C09106=1036.501,256.965,387.007,171.006,42.916,158.201
C09107=1036.494,256.716,387.037,171.003,42.915,158.201
C09108=1036.487,256.469,387.066,171.000,42.914,158.200
C09109=1036.480,256.220,387.095,170.997,42.914,158.200
C09110=1036.474,255.973,387.125,170.993,42.913,158.200
C09111=1036.468,255.724,387.154,170.991,42.912,158.199
C09112=1036.461,255.476,387.183,170.987,42.911,158.199
C09113=1036.454,255.228,387.213,170.985,42.910,158.198
C09114=1036.447,254.979,387.242,170.981,42.910,158.198
C09115=1036.441,254.731,387.272,170.978,42.909,158.198
C09116=1036.433,254.483,387.301,170.976,42.908,158.197
C09117=1036.427,254.235,387.330,170.972,42.907,158.197
C09118=1036.420,253.987,387.360,170.969,42.907,158.196
C09119=1036.413,253.739,387.389,170.966,42.906,158.196
C09120=1036.407,253.490,387.419,170.963,42.905,158.196
C09121=1036.400,253.242,387.448,170.960,42.903,158.195
C09122=1036.394,252.994,387.477,170.957,42.903,158.195
C09123=1036.387,252.745,387.507,170.953,42.902,158.194
C09124=1036.380,252.498,387.535,170.951,42.901,158.194
C09125=1036.373,252.249,387.565,170.947,42.900,158.193
C09126=1036.367,252.001,387.594,170.945,42.899,158.193
C09127=1036.360,251.753,387.624,170.941,42.899,158.193
C09128=1036.353,251.504,387.653,170.938,42.898,158.192
C09129=1036.347,251.256,387.682,170.936,42.897,158.192
C09130=1036.340,251.009,387.711,170.932,42.896,158.191
C09131=1036.333,250.760,387.741,170.930,42.895,158.191
C09132=1036.327,250.512,387.770,170.926,42.895,158.191
C09133=1036.321,250.264,387.799,170.924,42.894,158.190
C09134=1036.314,250.015,387.828,170.920,42.893,158.190
C09135=1036.307,249.767,387.857,170.917,42.892,158.189
C09136=1036.301,249.519,387.887,170.914,42.891,158.189
C09137=1036.291,249.191,387.924,170.911,42.890,158.189
C09138=1036.283,248.864,387.963,170.906,42.889,158.188
C09139=1036.274,248.536,388.001,170.903,42.888,158.187
C09140=1036.266,248.209,388.040,170.899,42.887,158.187
C09141=1036.259,247.960,388.069,170.896,42.886,158.187
C09142=1036.253,247.712,388.098,170.892,42.885,158.186
C09143=1036.246,247.464,388.127,170.890,42.884,158.186
C09144=1036.240,247.216,388.156,170.886,42.884,158.185
C09145=1036.233,246.967,388.185,170.884,42.883,158.185
C09146=1036.226,246.719,388.214,170.880,42.882,158.185
C09147=1036.220,246.471,388.243,170.878,42.881,158.184
C09148=1036.214,246.223,388.272,170.874,42.880,158.184
C09149=1036.207,245.974,388.302,170.872,42.879,158.183
C09150=1036.200,245.726,388.330,170.869,42.879,158.183
C09151=1036.194,245.478,388.359,170.866,42.878,158.183
C09152=1036.188,245.230,388.388,170.863,42.877,158.182
C09153=1036.181,244.982,388.417,170.860,42.876,158.182
C09154=1036.174,244.733,388.447,170.858,42.875,158.181
C09155=1036.167,244.485,388.475,170.854,42.874,158.181
C09156=1036.161,244.237,388.504,170.852,42.874,158.181
C09157=1036.155,243.988,388.532,170.849,42.873,158.180
C09158=1036.148,243.740,388.561,170.846,42.873,158.180
C09159=1036.141,243.492,388.590,170.843,42.872,158.180
C09160=1036.134,243.244,388.619,170.840,42.871,158.179
C09161=1036.128,242.995,388.648,170.837,42.870,158.179
C09162=1036.122,242.747,388.676,170.834,42.869,158.178
C09163=1036.115,242.498,388.705,170.831,42.868,158.178
C09164=1036.108,242.250,388.734,170.829,42.868,158.178
C09165=1036.101,242.002,388.763,170.825,42.867,158.177
C09166=1036.095,241.754,388.790,170.823,42.867,158.177
C09167=1036.089,241.506,388.819,170.819,42.866,158.177
C09168=1036.082,241.258,388.848,170.817,42.865,158.176
C09169=1036.075,241.008,388.877,170.814,42.864,158.176
C09170=1036.068,240.761,388.905,170.811,42.863,158.175
C09171=1036.062,240.512,388.934,170.808,42.863,158.175
C09172=1036.055,240.264,388.962,170.805,42.862,158.175
C09173=1036.048,240.016,388.990,170.802,42.861,158.174
C09174=1036.042,239.767,389.018,170.800,42.861,158.174
C09175=1036.035,239.519,389.047,170.796,42.860,158.174
C09176=1036.028,239.271,389.076,170.794,42.860,158.173
C09177=1036.022,239.022,389.104,170.791,42.859,158.173
C09178=1036.015,238.775,389.133,170.788,42.858,158.173
C09179=1036.008,238.526,389.160,170.786,42.857,158.172
C09180=1036.002,238.278,389.189,170.782,42.857,158.172
C09181=1035.995,238.030,389.217,170.780,42.856,158.172
C09182=1035.987,237.781,389.246,170.776,42.855,158.171
C09183=1035.981,237.532,389.274,170.774,42.854,158.171
C09184=1035.974,237.284,389.303,170.771,42.854,158.170
C09185=1035.968,237.036,389.330,170.768,42.853,158.170
C09186=1035.961,236.788,389.358,170.766,42.852,158.170
C09187=1035.955,236.539,389.387,170.762,42.852,158.169
C09188=1035.948,236.291,389.415,170.760,42.851,158.169
C09189=1035.941,236.043,389.443,170.757,42.851,158.169
C09190=1035.935,235.795,389.471,170.754,42.850,158.168
C09191=1035.927,235.546,389.499,170.751,42.849,158.168
C09192=1035.921,235.297,389.528,170.749,42.849,158.168
C09193=1035.912,234.964,389.565,170.745,42.847,158.167
C09194=1035.903,234.631,389.603,170.742,42.846,158.167
C09195=1035.894,234.297,389.641,170.737,42.846,158.166
C09196=1035.885,233.964,389.679,170.734,42.845,158.166
C09197=1035.879,233.715,389.707,170.731,42.844,158.165
C09198=1035.872,233.467,389.735,170.728,42.844,158.165
C09199=1035.865,233.219,389.763,170.725,42.843,158.165
C09200=1035.859,232.970,389.791,170.723,42.842,158.164
C09201=1035.852,232.722,389.819,170.720,42.842,158.164
C09202=1035.846,232.474,389.848,170.717,42.841,158.164
C09203=1035.839,232.225,389.875,170.714,42.841,158.163
C09204=1035.832,231.977,389.903,170.712,42.840,158.163
C09205=1035.826,231.728,389.931,170.709,42.839,158.163
C09206=1035.819,231.481,389.959,170.706,42.838,158.162
C09207=1035.812,231.232,389.987,170.703,42.838,158.162
C09208=1035.806,230.983,390.015,170.701,42.837,158.162
C09209=1035.799,230.735,390.043,170.698,42.836,158.161
C09210=1035.793,230.487,390.071,170.695,42.836,158.161
C09211=1035.786,230.238,390.099,170.693,42.835,158.161
C09212=1035.779,229.990,390.126,170.690,42.835,158.160
C09213=1035.773,229.741,390.154,170.687,42.834,158.160
C09214=1035.766,229.493,390.183,170.685,42.833,158.160
C09215=1035.759,229.245,390.210,170.681,42.833,158.159
C09216=1035.752,228.997,390.238,170.679,42.832,158.159
C09217=1035.746,228.748,390.266,170.677,42.831,158.159
C09218=1035.739,228.500,390.293,170.673,42.831,158.158
C09219=1035.732,228.251,390.321,170.671,42.830,158.158
C09220=1035.726,228.003,390.349,170.669,42.829,158.158
C09221=1035.719,227.754,390.377,170.665,42.829,158.157
C09222=1035.712,227.506,390.404,170.663,42.828,158.157
C09223=1035.706,227.257,390.432,170.660,42.828,158.157
C09224=1035.699,227.009,390.460,170.657,42.827,158.156
C09225=1035.692,226.762,390.487,170.655,42.827,158.156
C09226=1035.685,226.513,390.514,170.651,42.826,158.156
C09227=1035.679,226.265,390.542,170.649,42.825,158.155
C09228=1035.672,226.016,390.569,170.647,42.825,158.155
C09229=1035.666,225.767,390.597,170.643,42.824,158.155
C09230=1035.659,225.519,390.625,170.641,42.824,158.154
C09231=1035.652,225.271,390.652,170.639,42.823,158.154
C09232=1035.645,225.022,390.679,170.636,42.822,158.154
C09233=1035.638,224.774,390.707,170.633,42.822,158.153
C09234=1035.631,224.525,390.735,170.631,42.821,158.153
C09235=1035.625,224.276,390.762,170.628,42.820,158.153
C09236=1035.618,224.028,390.790,170.625,42.820,158.153
C09237=1035.612,223.780,390.816,170.623,42.819,158.152
C09238=1035.605,223.532,390.844,170.620,42.818,158.152
C09239=1035.598,223.283,390.872,170.617,42.818,158.152
C09240=1035.592,223.035,390.900,170.615,42.817,158.151
C09241=1035.585,222.786,390.927,170.612,42.817,158.151
C09242=1035.579,222.538,390.954,170.610,42.816,158.151
C09243=1035.571,222.289,390.981,170.607,42.816,158.150
C09244=1035.565,222.042,391.009,170.604,42.815,158.150
C09245=1035.559,221.793,391.036,170.602,42.815,158.150
C09246=1035.552,221.544,391.064,170.600,42.814,158.149
C09247=1035.545,221.296,391.091,170.596,42.814,158.149
C09248=1035.538,221.048,391.118,170.594,42.813,158.149
C09249=1035.529,220.706,391.156,170.590,42.812,158.148
C09250=1035.520,220.365,391.194,170.587,42.811,158.148
C09251=1035.511,220.024,391.230,170.584,42.811,158.147
C09252=1035.502,219.684,391.268,170.580,42.809,158.147
C09253=1035.495,219.435,391.295,170.577,42.809,158.147
C09254=1035.489,219.186,391.322,170.574,42.809,158.146
C09255=1035.482,218.938,391.350,170.572,42.808,158.146
C09256=1035.475,218.689,391.377,170.570,42.808,158.146
C09257=1035.468,218.442,391.403,170.566,42.807,158.145
C09258=1035.462,218.192,391.430,170.564,42.806,158.145
C09259=1035.455,217.944,391.458,170.562,42.806,158.145
C09260=1035.448,217.695,391.485,170.559,42.805,158.145
C09261=1035.441,217.447,391.512,170.556,42.805,158.144
C09262=1035.435,217.199,391.538,170.554,42.804,158.144
C09263=1035.428,216.951,391.565,170.552,42.804,158.144
C09264=1035.421,216.702,391.592,170.549,42.803,158.143
C09265=1035.414,216.453,391.620,170.546,42.803,158.143
C09266=1035.408,216.205,391.646,170.543,42.802,158.143
C09267=1035.401,215.957,391.674,170.541,42.802,158.142
C09268=1035.394,215.708,391.700,170.539,42.801,158.142
C09269=1035.388,215.459,391.728,170.537,42.800,158.142
C09270=1035.381,215.211,391.754,170.533,42.800,158.142
C09271=1035.374,214.963,391.782,170.531,42.799,158.141
C09272=1035.367,214.714,391.808,170.529,42.799,158.141
C09273=1035.361,214.465,391.835,170.526,42.798,158.141
C09274=1035.354,214.218,391.862,170.524,42.798,158.140
C09275=1035.348,213.969,391.889,170.521,42.797,158.140
C09276=1035.341,213.720,391.916,170.518,42.797,158.140
C09277=1035.334,213.472,391.943,170.516,42.796,158.140
C09278=1035.327,213.223,391.969,170.514,42.796,158.139
C09279=1035.321,212.975,391.997,170.511,42.795,158.139
C09280=1035.314,212.726,392.024,170.508,42.794,158.139
C09281=1035.308,212.478,392.050,170.506,42.794,158.138
C09282=1035.300,212.230,392.077,170.503,42.793,158.138
C09283=1035.294,211.981,392.104,170.501,42.793,158.138
C09284=1035.287,211.733,392.130,170.499,42.792,158.137
C09285=1035.281,211.484,392.157,170.496,42.792,158.137
C09286=1035.274,211.235,392.185,170.493,42.791,158.137
C09287=1035.268,210.987,392.211,170.491,42.791,158.136
C09288=1035.261,210.738,392.238,170.489,42.790,158.136
C09289=1035.254,210.490,392.264,170.486,42.789,158.136
C09290=1035.248,210.242,392.291,170.484,42.789,158.136
C09291=1035.240,209.993,392.318,170.482,42.789,158.135
C09292=1035.233,209.744,392.344,170.478,42.788,158.135
C09293=1035.228,209.496,392.371,170.476,42.788,158.135
C09294=1035.220,209.247,392.397,170.474,42.787,158.134
C09295=1035.214,208.999,392.423,170.471,42.787,158.134
C09296=1035.207,208.751,392.451,170.469,42.786,158.134
C09297=1035.200,208.502,392.477,170.467,42.785,158.134
C09298=1035.194,208.254,392.504,170.464,42.785,158.133
C09299=1035.187,208.005,392.530,170.461,42.785,158.133
C09300=1035.180,207.756,392.557,170.459,42.784,158.133
C09301=1035.174,207.508,392.583,170.456,42.784,158.133
C09302=1035.167,207.259,392.609,170.454,42.783,158.132
C09303=1035.160,207.011,392.635,170.452,42.782,158.132
C09304=1035.154,206.762,392.663,170.450,42.782,158.132
C09305=1035.144,206.427,392.698,170.446,42.781,158.131
C09306=1035.135,206.092,392.733,170.443,42.781,158.131
C09307=1035.125,205.756,392.769,170.439,42.781,158.131
C09308=1035.117,205.421,392.805,170.436,42.780,158.130
C09309=1035.090,204.371,392.911,170.114,42.675,158.085
C09310=1035.085,204.123,392.935,170.111,42.676,158.085
C09311=1035.079,203.874,392.961,170.108,42.675,158.085
C09312=1035.073,203.625,392.986,170.105,42.676,158.085
C09313=1035.066,203.377,393.011,170.101,42.677,158.085
C09314=1035.059,203.128,393.036,170.097,42.676,158.084
C09315=1035.054,202.879,393.061,170.094,42.677,158.084
C09316=1035.048,202.631,393.086,170.091,42.677,158.084
C09317=1035.042,202.382,393.111,170.088,42.677,158.084
C09318=1035.036,202.133,393.136,170.084,42.678,158.084
C09319=1035.030,201.884,393.161,170.081,42.678,158.083
C09320=1035.023,201.636,393.186,170.078,42.678,158.083
C09321=1035.018,201.388,393.211,170.075,42.678,158.083
C09322=1035.012,201.138,393.236,170.071,42.679,158.083
C09323=1035.005,200.890,393.261,170.067,42.679,158.083
C09324=1034.999,200.641,393.285,170.064,42.679,158.083
C09325=1034.993,200.392,393.311,170.061,42.680,158.082
C09326=1034.987,200.144,393.334,170.058,42.680,158.082
C09327=1034.981,199.895,393.360,170.054,42.681,158.082
C09328=1034.974,199.647,393.384,170.051,42.681,158.082
C09329=1034.968,199.397,393.409,170.048,42.681,158.082
C09330=1034.962,199.148,393.434,170.045,42.682,158.082
C09331=1034.956,198.901,393.458,170.042,42.682,158.082
C09332=1034.950,198.651,393.483,170.038,42.683,158.081
C09333=1034.943,198.403,393.507,170.035,42.683,158.081
C09334=1034.937,198.154,393.532,170.031,42.683,158.081
C09335=1034.930,197.905,393.557,170.028,42.683,158.081
C09336=1034.925,197.657,393.581,170.025,42.684,158.081
C09337=1034.918,197.408,393.606,170.021,42.685,158.081
C09338=1034.912,197.159,393.630,170.018,42.685,158.080
C09339=1034.905,196.910,393.654,170.015,42.686,158.080
C09340=1034.899,196.662,393.679,170.012,42.685,158.080
C09341=1034.893,196.413,393.703,170.009,42.686,158.080
C09342=1034.887,196.164,393.728,170.005,42.687,158.080
C09343=1034.881,195.916,393.752,170.002,42.687,158.080
C09344=1034.875,195.667,393.777,169.999,42.688,158.080
C09345=1034.868,195.418,393.801,169.996,42.688,158.079
C09346=1034.862,195.170,393.826,169.993,42.689,158.079
C09347=1034.856,194.921,393.850,169.990,42.689,158.079
C09348=1034.850,194.672,393.875,169.985,42.689,158.079
C09349=1034.844,194.424,393.900,169.982,42.690,158.079
C09350=1034.838,194.175,393.924,169.979,42.690,158.079
C09351=1034.832,193.925,393.948,169.976,42.691,158.079
C09352=1034.826,193.677,393.972,169.973,42.691,158.078
C09353=1034.819,193.428,393.997,169.970,42.692,158.078
C09354=1034.813,193.179,394.021,169.967,42.692,158.078
C09355=1034.808,192.931,394.046,169.963,42.693,158.078
C09356=1034.801,192.682,394.070,169.960,42.693,158.078
C09357=1034.795,192.433,394.094,169.957,42.694,158.078
C09358=1034.789,192.185,394.119,169.954,42.693,158.078
C09359=1034.783,191.936,394.143,169.951,42.694,158.077
C09360=1034.777,191.687,394.167,169.948,42.694,158.077
C09361=1034.770,191.438,394.191,169.945,42.695,158.077
C09362=1034.765,191.190,394.215,169.942,42.695,158.077
C09363=1034.758,190.941,394.239,169.939,42.696,158.077
C09364=1034.752,190.692,394.264,169.935,42.697,158.077
C09365=1034.746,190.444,394.288,169.932,42.697,158.077
C09366=1034.740,190.195,394.313,169.928,42.698,158.077
C09367=1034.734,189.946,394.336,169.925,42.698,158.076
C09368=1034.728,189.697,394.361,169.922,42.699,158.076
C09369=1034.722,189.449,394.385,169.919,42.699,158.076
C09370=1034.715,189.165,394.413,169.915,42.700,158.076
C09371=1034.708,188.880,394.440,169.912,42.700,158.076
C09372=1034.701,188.597,394.468,169.909,42.701,158.076
C09373=1034.694,188.312,394.495,169.905,42.701,158.076
C09374=1034.689,188.063,394.519,169.902,42.702,158.076
C09375=1034.682,187.814,394.543,169.899,42.702,158.075
C09376=1034.677,187.566,394.567,169.896,42.702,158.075
C09377=1034.671,187.317,394.591,169.893,42.703,158.075
C09378=1034.665,187.068,394.616,169.890,42.703,158.075
C09379=1034.659,186.819,394.640,169.887,42.704,158.075
C09380=1034.653,186.571,394.664,169.884,42.704,158.075
C09381=1034.647,186.322,394.688,169.881,42.705,158.075
C09382=1034.641,186.073,394.712,169.878,42.705,158.074
C09383=1034.635,185.825,394.736,169.875,42.706,158.074
C09384=1034.629,185.576,394.760,169.872,42.706,158.074
C09385=1034.623,185.327,394.784,169.869,42.707,158.074
C09386=1034.617,185.078,394.808,169.865,42.707,158.074
C09387=1034.611,184.830,394.833,169.862,42.708,158.074
C09388=1034.605,184.582,394.856,169.859,42.708,158.074
C09389=1034.600,184.332,394.880,169.856,42.709,158.074
C09390=1034.594,184.083,394.904,169.853,42.709,158.073
C09391=1034.588,183.834,394.928,169.850,42.709,158.073
C09392=1034.582,183.586,394.952,169.847,42.710,158.073
C09393=1034.576,183.338,394.976,169.844,42.710,158.073
C09394=1034.570,183.088,395.000,169.841,42.712,158.073
C09395=1034.564,182.839,395.023,169.838,42.712,158.073
C09396=1034.557,182.591,395.047,169.834,42.713,158.073
C09397=1034.551,182.342,395.070,169.831,42.713,158.073
C09398=1034.544,182.093,395.094,169.828,42.714,158.073
C09399=1034.539,181.844,395.117,169.825,42.715,158.073
C09400=1034.532,181.595,395.141,169.822,42.715,158.073
C09401=1034.526,181.347,395.164,169.819,42.716,158.073
C09402=1034.520,181.097,395.188,169.816,42.717,158.072
C09403=1034.514,180.849,395.211,169.813,42.717,158.072
C09404=1034.507,180.600,395.234,169.811,42.719,158.072
C09405=1034.501,180.351,395.258,169.808,42.719,158.072
C09406=1034.495,180.102,395.281,169.804,42.720,158.072
C09407=1034.488,179.853,395.305,169.802,42.721,158.072
C09408=1034.482,179.604,395.328,169.799,42.721,158.072
C09409=1034.476,179.356,395.351,169.796,42.722,158.072
C09410=1034.470,179.107,395.375,169.793,42.723,158.072
C09411=1034.463,178.859,395.398,169.790,42.723,158.072
C09412=1034.457,178.609,395.421,169.787,42.724,158.072
C09413=1034.451,178.361,395.445,169.784,42.725,158.072
C09414=1034.445,178.112,395.468,169.781,42.725,158.072
C09415=1034.439,177.863,395.492,169.778,42.727,158.072
C09416=1034.433,177.614,395.515,169.775,42.727,158.072
C09417=1034.426,177.365,395.537,169.772,42.728,158.071
C09418=1034.420,177.116,395.561,169.769,42.729,158.071
C09419=1034.414,176.867,395.584,169.766,42.729,158.071
C09420=1034.408,176.619,395.608,169.763,42.730,158.071
C09421=1034.402,176.370,395.631,169.760,42.731,158.071
C09422=1034.396,176.121,395.654,169.757,42.731,158.071
C09423=1034.390,175.872,395.677,169.754,42.732,158.071
C09424=1034.383,175.623,395.700,169.751,42.733,158.071
C09425=1034.377,175.374,395.723,169.748,42.733,158.071
C09426=1034.371,175.126,395.747,169.745,42.735,158.071
C09427=1034.365,174.876,395.770,169.742,42.735,158.071
C09428=1034.359,174.627,395.793,169.739,42.735,158.071
C09429=1034.353,174.379,395.817,169.736,42.737,158.071
C09430=1034.346,174.131,395.839,169.733,42.737,158.071
C09431=1034.340,173.881,395.862,169.730,42.738,158.071
C09432=1034.334,173.633,395.886,169.727,42.739,158.070
C09433=1034.328,173.384,395.909,169.724,42.739,158.070
C09434=1034.321,173.099,395.935,169.722,42.740,158.070
C09435=1034.314,172.815,395.962,169.718,42.741,158.070
C09436=1034.308,172.530,395.988,169.715,42.742,158.070
C09437=1034.300,172.246,396.014,169.712,42.743,158.070
C09438=1034.295,171.997,396.037,169.709,42.744,158.070
C09439=1034.288,171.748,396.060,169.706,42.744,158.070
C09440=1034.282,171.499,396.084,169.703,42.745,158.070
C09441=1034.276,171.251,396.106,169.700,42.746,158.070
C09442=1034.270,171.002,396.129,169.697,42.746,158.070
C09443=1034.264,170.753,396.152,169.694,42.748,158.070
C09444=1034.258,170.503,396.176,169.691,42.748,158.070
C09445=1034.252,170.255,396.198,169.688,42.749,158.070
C09446=1034.246,170.006,396.222,169.685,42.750,158.070
C09447=1034.240,169.758,396.244,169.682,42.750,158.069
C09448=1034.234,169.509,396.267,169.680,42.751,158.070
C09449=1034.228,169.260,396.290,169.677,42.752,158.069
C09450=1034.222,169.010,396.314,169.674,42.752,158.069
C09451=1034.215,168.762,396.336,169.671,42.753,158.069
C09452=1034.210,168.513,396.359,169.668,42.754,158.069
C09453=1034.204,168.264,396.382,169.665,42.755,158.069
C09454=1034.198,168.015,396.405,169.662,42.755,158.069
C09455=1034.193,167.766,396.428,169.659,42.756,158.069
C09456=1034.186,167.518,396.450,169.656,42.757,158.069
C09457=1034.180,167.269,396.474,169.654,42.757,158.069
C09458=1034.174,167.020,396.497,169.652,42.758,158.069
C09459=1034.168,166.771,396.520,169.649,42.759,158.069
C09460=1034.162,166.522,396.543,169.646,42.760,158.069
C09461=1034.156,166.273,396.565,169.643,42.761,158.069
C09462=1034.150,166.024,396.588,169.640,42.761,158.069
C09463=1034.144,165.776,396.611,169.637,42.762,158.069
C09464=1034.139,165.527,396.634,169.635,42.763,158.069
C09465=1034.132,165.278,396.657,169.632,42.764,158.069
C09466=1034.127,165.029,396.679,169.629,42.764,158.068
C09467=1034.121,164.780,396.702,169.626,42.765,158.068
C09468=1034.115,164.531,396.725,169.623,42.766,158.068
C09469=1034.110,164.282,396.748,169.620,42.766,158.068
C09470=1034.103,164.033,396.770,169.618,42.767,158.068
C09471=1034.097,163.784,396.793,169.615,42.768,158.068
C09472=1034.092,163.535,396.816,169.612,42.769,158.068
C09473=1034.086,163.287,396.839,169.609,42.769,158.068
C09474=1034.079,163.038,396.861,169.606,42.770,158.068
C09475=1034.074,162.789,396.884,169.604,42.771,158.068
C09476=1034.068,162.540,396.907,169.601,42.771,158.068
C09477=1034.063,162.291,396.929,169.599,42.772,158.068
C09478=1034.056,162.042,396.952,169.595,42.773,158.068
C09479=1034.050,161.793,396.975,169.593,42.774,158.068
C09480=1034.045,161.544,396.998,169.591,42.774,158.068
C09481=1034.039,161.295,397.020,169.588,42.776,158.068
C09482=1034.032,161.047,397.043,169.585,42.776,158.068
C09483=1034.027,160.797,397.065,169.582,42.777,158.068
C09484=1034.021,160.548,397.088,169.579,42.778,158.067
C09485=1034.015,160.300,397.111,169.577,42.778,158.067
C09486=1034.009,160.051,397.133,169.574,42.779,158.067
C09487=1034.004,159.801,397.156,169.571,42.780,158.067
C09488=1033.997,159.553,397.178,169.568,42.781,158.067
C09489=1033.991,159.304,397.201,169.565,42.782,158.067
C09490=1033.985,159.055,397.222,169.563,42.782,158.067
C09491=1033.979,158.806,397.245,169.560,42.783,158.067
C09492=1033.973,158.557,397.268,169.558,42.785,158.067
C09493=1033.967,158.308,397.289,169.554,42.785,158.067
C09494=1033.960,158.059,397.312,169.552,42.786,158.067
C09495=1033.955,157.810,397.334,169.549,42.787,158.067
C09496=1033.949,157.561,397.356,169.547,42.788,158.067
C09497=1033.942,157.312,397.378,169.544,42.789,158.067
C09498=1033.935,157.028,397.404,169.541,42.790,158.067
C09499=1033.929,156.743,397.429,169.537,42.791,158.067
C09500=1033.922,156.458,397.454,169.534,42.792,158.067
C09501=1033.915,156.173,397.480,169.531,42.793,158.067
C09502=1033.908,155.924,397.502,169.529,42.794,158.067
C09503=1033.903,155.675,397.525,169.525,42.794,158.067
C09504=1033.897,155.426,397.546,169.524,42.795,158.067
C09505=1033.891,155.178,397.569,169.521,42.797,158.067
C09506=1033.885,154.928,397.591,169.518,42.797,158.067
C09507=1033.879,154.680,397.613,169.515,42.798,158.067
C09508=1033.873,154.430,397.635,169.512,42.799,158.067
C09509=1033.867,154.182,397.658,169.510,42.800,158.067
C09510=1033.861,153.932,397.679,169.507,42.801,158.067
C09511=1033.854,153.683,397.701,169.504,42.802,158.067
C09512=1033.848,153.435,397.723,169.502,42.803,158.067
C09513=1033.842,153.185,397.745,169.499,42.804,158.067
C09514=1033.836,152.936,397.768,169.497,42.805,158.067
C09515=1033.831,152.688,397.789,169.494,42.806,158.067
C09516=1033.824,152.439,397.811,169.491,42.807,158.067
C09517=1033.818,152.190,397.833,169.488,42.807,158.067
C09518=1033.812,151.941,397.855,169.485,42.808,158.067
C09519=1033.806,151.692,397.876,169.483,42.809,158.067
C09520=1033.800,151.443,397.899,169.480,42.811,158.067
C09521=1033.794,151.194,397.921,169.477,42.811,158.067
C09522=1033.788,150.944,397.943,169.475,42.812,158.067
C09523=1033.782,150.697,397.965,169.473,42.813,158.067
C09524=1033.776,150.447,397.986,169.470,42.814,158.067
C09525=1033.769,150.198,398.008,169.467,42.815,158.067
C09526=1033.764,149.949,398.030,169.464,42.816,158.067
C09527=1033.757,149.700,398.052,169.462,42.817,158.067
C09528=1033.751,149.451,398.074,169.459,42.818,158.067
C09529=1033.746,149.202,398.095,169.456,42.819,158.067
C09530=1033.740,148.953,398.117,169.453,42.820,158.067
C09531=1033.733,148.705,398.139,169.452,42.821,158.067
C09532=1033.727,148.455,398.161,169.449,42.822,158.067
C09533=1033.721,148.206,398.183,169.446,42.822,158.067
C09534=1033.715,147.958,398.204,169.443,42.823,158.067
C09535=1033.710,147.708,398.226,169.441,42.824,158.067
C09536=1033.704,147.459,398.248,169.438,42.826,158.067
C09537=1033.697,147.210,398.270,169.435,42.827,158.067
C09538=1033.691,146.961,398.292,169.432,42.827,158.067
C09539=1033.685,146.713,398.313,169.431,42.828,158.067
C09540=1033.679,146.463,398.335,169.428,42.829,158.067
C09541=1033.673,146.214,398.356,169.425,42.831,158.067
C09542=1033.667,145.965,398.378,169.422,42.832,158.067
C09543=1033.660,145.716,398.399,169.420,42.833,158.067
C09544=1033.654,145.468,398.420,169.417,42.833,158.067
C09545=1033.648,145.218,398.442,169.414,42.834,158.067
C09546=1033.642,144.969,398.464,169.411,42.835,158.067
C09547=1033.636,144.720,398.485,169.410,42.836,158.067
C09548=1033.630,144.471,398.507,169.407,42.838,158.067
C09549=1033.624,144.222,398.528,169.404,42.839,158.067
C09550=1033.618,143.973,398.550,169.401,42.840,158.067
C09551=1033.612,143.724,398.571,169.399,42.841,158.067
C09552=1033.605,143.475,398.592,169.396,42.841,158.067
C09553=1033.599,143.226,398.614,169.393,42.842,158.067
C09554=1033.593,142.977,398.635,169.392,42.843,158.067
C09555=1033.587,142.728,398.657,169.389,42.845,158.067
C09556=1033.581,142.479,398.679,169.386,42.846,158.067
C09557=1033.575,142.230,398.700,169.383,42.847,158.067
C09558=1033.569,141.981,398.721,169.381,42.848,158.067
C09559=1033.563,141.732,398.743,169.378,42.848,158.067
C09560=1033.558,141.483,398.764,169.375,42.849,158.067
C09561=1033.551,141.235,398.785,169.374,42.850,158.067
C09562=1033.543,140.886,398.815,169.370,42.852,158.067
C09563=1033.534,140.536,398.846,169.366,42.854,158.067
C09564=1033.525,140.188,398.875,169.362,42.855,158.067
C09565=1033.517,139.839,398.905,169.358,42.856,158.067
C09566=1033.511,139.590,398.926,169.356,42.857,158.067
C09567=1033.505,139.341,398.948,169.354,42.858,158.067
C09568=1033.499,139.092,398.969,169.351,42.860,158.067
C09569=1033.493,138.843,398.991,169.349,42.861,158.067
C09570=1033.486,138.594,399.012,169.346,42.861,158.067
C09571=1033.481,138.345,399.033,169.343,42.862,158.067
C09572=1033.475,138.096,399.054,169.341,42.863,158.067
C09573=1033.468,137.847,399.075,169.338,42.864,158.067
C09574=1033.462,137.598,399.097,169.336,42.866,158.067
C09575=1033.457,137.348,399.117,169.333,42.867,158.067
C09576=1033.450,137.100,399.138,169.331,42.868,158.067
C09577=1033.444,136.851,399.160,169.328,42.869,158.067
C09578=1033.438,136.602,399.181,169.325,42.870,158.067
C09579=1033.433,136.353,399.202,169.323,42.871,158.067
C09580=1033.426,136.104,399.223,169.321,42.872,158.067
C09581=1033.420,135.855,399.245,169.318,42.873,158.067
C09582=1033.414,135.606,399.265,169.316,42.874,158.067
C09583=1033.408,135.357,399.286,169.313,42.875,158.067
C09584=1033.401,135.107,399.308,169.310,42.876,158.067
C09585=1033.395,134.859,399.328,169.308,42.877,158.067
C09586=1033.389,134.609,399.349,169.306,42.879,158.067
C09587=1033.384,134.360,399.370,169.303,42.880,158.067
C09588=1033.377,134.111,399.391,169.301,42.881,158.068
C09589=1033.371,133.862,399.413,169.298,42.882,158.068
C09590=1033.365,133.613,399.433,169.295,42.883,158.068
C09591=1033.359,133.364,399.454,169.293,42.884,158.068
C09592=1033.353,133.115,399.475,169.291,42.885,158.068
C09593=1033.347,132.866,399.496,169.288,42.886,158.068
C09594=1033.340,132.617,399.517,169.286,42.887,158.068
C09595=1033.334,132.368,399.537,169.283,42.888,158.068
C09596=1033.328,132.119,399.559,169.280,42.890,158.068
C09597=1033.323,131.870,399.580,169.278,42.890,158.068
C09598=1033.316,131.621,399.601,169.275,42.891,158.068
C09599=1033.311,131.372,399.621,169.272,42.892,158.068
C09600=1033.304,131.123,399.642,169.271,42.893,158.068
C09601=1033.299,130.874,399.663,169.268,42.894,158.068
C09602=1033.293,130.625,399.684,169.265,42.896,158.068
C09603=1033.286,130.375,399.705,169.263,42.896,158.068
C09604=1033.280,130.127,399.725,169.260,42.898,158.068
C09605=1033.273,129.877,399.746,169.258,42.899,158.068
C09606=1033.268,129.628,399.766,169.256,42.900,158.068
C09607=1033.261,129.379,399.787,169.253,42.902,158.068
C09608=1033.255,129.131,399.807,169.250,42.903,158.068
C09609=1033.249,128.881,399.829,169.248,42.904,158.068
C09610=1033.242,128.632,399.849,169.245,42.905,158.068
C09611=1033.236,128.383,399.869,169.243,42.906,158.068
C09612=1033.229,128.134,399.890,169.240,42.908,158.068
C09613=1033.224,127.885,399.911,169.238,42.909,158.068
C09614=1033.217,127.635,399.931,169.235,42.910,158.068
C09615=1033.211,127.387,399.952,169.232,42.911,158.068
C09616=1033.205,127.137,399.973,169.231,42.912,158.068
C09617=1033.199,126.889,399.993,169.228,42.913,158.068
C09618=1033.192,126.640,400.014,169.225,42.914,158.068
C09619=1033.186,126.391,400.034,169.223,42.915,158.069
C09620=1033.180,126.141,400.055,169.221,42.917,158.069
C09621=1033.174,125.892,400.075,169.218,42.918,158.069
C09622=1033.165,125.521,400.105,169.215,42.919,158.069
C09623=1033.156,125.150,400.136,169.211,42.921,158.069
C09624=1033.149,124.865,400.160,169.208,42.923,158.069
C09625=1033.142,124.579,400.183,169.205,42.924,158.069
C09626=1033.135,124.295,400.206,169.203,42.926,158.069
C09627=1033.128,124.010,400.230,169.199,42.927,158.069
C09628=1033.122,123.760,400.251,169.197,42.928,158.069
C09629=1033.116,123.511,400.271,169.194,42.929,158.069
C09630=1033.109,123.261,400.291,169.193,42.930,158.069
C09631=1033.103,123.013,400.312,169.190,42.931,158.069
C09632=1033.097,122.763,400.332,169.187,42.932,158.069
C09633=1033.091,122.515,400.352,169.185,42.934,158.069
C09634=1033.085,122.266,400.372,169.182,42.935,158.069
C09635=1033.078,122.016,400.393,169.180,42.936,158.069
C09636=1033.073,121.767,400.413,169.178,42.937,158.069
C09637=1033.067,121.518,400.434,169.175,42.938,158.069
C09638=1033.060,121.269,400.454,169.173,42.939,158.069
C09639=1033.054,121.021,400.474,169.170,42.941,158.069
C09640=1033.048,120.771,400.495,169.167,42.942,158.070
C09641=1033.042,120.522,400.515,169.166,42.943,158.070
C09642=1033.036,120.272,400.535,169.163,42.944,158.070
C09643=1033.030,120.024,400.555,169.161,42.945,158.070
C09644=1033.025,119.774,400.576,169.158,42.947,158.070
C09645=1033.018,119.525,400.596,169.155,42.948,158.070
C09646=1033.012,119.276,400.616,169.154,42.949,158.070
C09647=1033.005,119.027,400.637,169.151,42.950,158.070
C09648=1033.000,118.778,400.658,169.149,42.951,158.070
C09649=1032.994,118.529,400.678,169.146,42.952,158.070
C09650=1032.987,118.280,400.698,169.143,42.953,158.070
C09651=1032.981,118.031,400.718,169.141,42.954,158.070
C09652=1032.975,117.782,400.738,169.139,42.955,158.070
C09653=1032.969,117.532,400.759,169.137,42.956,158.070
C09654=1032.963,117.284,400.779,169.134,42.957,158.070
C09655=1032.957,117.035,400.799,169.132,42.958,158.070
C09656=1032.951,116.785,400.819,169.129,42.960,158.070
C09657=1032.945,116.536,400.840,169.126,42.961,158.070
C09658=1032.940,116.287,400.860,169.125,42.962,158.070
C09659=1032.933,116.038,400.880,169.122,42.963,158.070
C09660=1032.927,115.789,400.900,169.120,42.964,158.070
C09661=1032.922,115.540,400.921,169.117,42.966,158.070
C09662=1032.916,115.291,400.940,169.115,42.967,158.070
C09663=1032.909,115.042,400.961,169.113,42.968,158.071
C09664=1032.903,114.792,400.980,169.110,42.969,158.071
C09665=1032.897,114.543,401.000,169.108,42.970,158.071
C09666=1032.892,114.293,401.021,169.105,42.971,158.071
C09667=1032.886,114.045,401.041,169.103,42.972,158.071
C09668=1032.880,113.796,401.061,169.100,42.973,158.071
C09669=1032.874,113.547,401.081,169.099,42.974,158.071
C09670=1032.868,113.297,401.102,169.096,42.975,158.071
C09671=1032.862,113.048,401.122,169.094,42.976,158.071
C09672=1032.856,112.800,401.142,169.091,42.978,158.071
C09673=1032.849,112.549,401.161,169.088,42.979,158.071
C09674=1032.843,112.301,401.181,169.086,42.980,158.071
C09675=1032.837,112.052,401.201,169.084,42.982,158.071
C09676=1032.831,111.803,401.221,169.082,42.983,158.071
C09677=1032.824,111.553,401.240,169.079,42.984,158.071
C09678=1032.818,111.304,401.260,169.076,42.985,158.071
C09679=1032.812,111.056,401.280,169.074,42.986,158.071
C09680=1032.806,110.806,401.300,169.072,42.987,158.071
C09681=1032.800,110.557,401.320,169.070,42.989,158.071
C09682=1032.794,110.308,401.340,169.067,42.990,158.071
C09683=1032.788,110.059,401.360,169.065,42.991,158.071
C09684=1032.782,109.809,401.379,169.062,42.992,158.071
C09685=1032.775,109.560,401.399,169.060,42.994,158.072
C09686=1032.769,109.312,401.418,169.058,42.995,158.072
C09687=1032.763,109.062,401.438,169.055,42.996,158.072
C09688=1032.756,108.777,401.461,169.052,42.997,158.072
C09689=1032.749,108.491,401.484,169.050,42.999,158.072
C09690=1032.742,108.205,401.506,169.047,43.000,158.072
C09691=1032.735,107.920,401.528,169.044,43.002,158.072
C09692=1032.729,107.671,401.548,169.042,43.003,158.072
C09693=1032.722,107.421,401.568,169.039,43.004,158.072
C09694=1032.716,107.173,401.588,169.037,43.005,158.072
C09695=1032.710,106.923,401.606,169.035,43.007,158.072
C09696=1032.704,106.675,401.626,169.032,43.008,158.072
C09697=1032.697,106.425,401.647,169.030,43.009,158.072
C09698=1032.692,106.176,401.666,169.028,43.010,158.072
C09699=1032.685,105.927,401.685,169.026,43.012,158.073
C09700=1032.679,105.678,401.704,169.023,43.013,158.073
C09701=1032.673,105.429,401.724,169.020,43.014,158.073
C09702=1032.667,105.179,401.744,169.018,43.015,158.073
C09703=1032.660,104.930,401.763,169.016,43.016,158.073
C09704=1032.655,104.681,401.783,169.014,43.018,158.073
C09705=1032.649,104.432,401.803,169.011,43.019,158.073
C09706=1032.643,104.183,401.822,169.009,43.020,158.073
C09707=1032.636,103.934,401.841,169.006,43.021,158.073
C09708=1032.630,103.684,401.861,169.005,43.022,158.073
C09709=1032.624,103.435,401.881,169.002,43.024,158.073
C09710=1032.618,103.186,401.900,168.999,43.025,158.073
C09711=1032.612,102.937,401.919,168.997,43.026,158.073
C09712=1032.606,102.688,401.939,168.994,43.027,158.073
C09713=1032.600,102.439,401.958,168.993,43.028,158.073
C09714=1032.594,102.190,401.978,168.990,43.030,158.073
C09715=1032.587,101.940,401.997,168.988,43.031,158.073
C09716=1032.581,101.691,402.017,168.985,43.032,158.073
C09717=1032.575,101.442,402.037,168.983,43.033,158.073
C09718=1032.569,101.193,402.056,168.981,43.034,158.073
C09719=1032.563,100.944,402.075,168.979,43.035,158.074
C09720=1032.557,100.695,402.095,168.976,43.037,158.074
C09721=1032.551,100.445,402.114,168.973,43.038,158.074
C09722=1032.546,100.196,402.133,168.972,43.039,158.074
C09723=1032.538,99.947,402.153,168.969,43.041,158.074
C09724=1032.533,99.697,402.172,168.967,43.042,158.074
C09725=1032.526,99.448,402.191,168.964,43.043,158.074
C09726=1032.520,99.199,402.211,168.962,43.044,158.074
C09727=1032.514,98.950,402.229,168.960,43.045,158.074
C09728=1032.508,98.701,402.248,168.957,43.047,158.074
C09729=1032.501,98.452,402.268,168.955,43.048,158.074
C09730=1032.496,98.203,402.287,168.952,43.049,158.074
C09731=1032.489,97.954,402.306,168.951,43.051,158.074
C09732=1032.483,97.704,402.325,168.948,43.052,158.074
C09733=1032.477,97.454,402.344,168.946,43.053,158.074
C09734=1032.471,97.206,402.364,168.943,43.055,158.075
C09735=1032.464,96.956,402.383,168.940,43.056,158.075
C09736=1032.458,96.707,402.402,168.939,43.057,158.075
C09737=1032.452,96.458,402.420,168.936,43.058,158.075
C09738=1032.445,96.209,402.440,168.934,43.060,158.075
C09739=1032.440,95.960,402.459,168.931,43.061,158.075
C09740=1032.433,95.711,402.478,168.930,43.062,158.075
C09741=1032.427,95.461,402.497,168.927,43.064,158.075
C09742=1032.421,95.212,402.516,168.925,43.065,158.075
C09743=1032.415,94.963,402.535,168.922,43.066,158.075
C09744=1032.409,94.714,402.554,168.919,43.067,158.075
C09745=1032.403,94.465,402.573,168.918,43.069,158.075
C09746=1032.396,94.216,402.592,168.915,43.070,158.075
C09747=1032.391,93.966,402.611,168.913,43.071,158.075
C09748=1032.384,93.717,402.630,168.910,43.073,158.076
C09749=1032.378,93.467,402.650,168.909,43.074,158.076
C09750=1032.372,93.218,402.668,168.906,43.075,158.076
C09751=1032.365,92.969,402.688,168.904,43.076,158.076
C09752=1032.358,92.684,402.709,168.901,43.078,158.076
C09753=1032.352,92.399,402.731,168.898,43.079,158.076
C09754=1032.344,92.113,402.753,168.896,43.081,158.076
C09755=1032.338,91.828,402.775,168.893,43.082,158.076
C09756=1032.331,91.578,402.793,168.891,43.083,158.076
C09757=1032.325,91.329,402.812,168.889,43.085,158.076
C09758=1032.319,91.080,402.831,168.886,43.086,158.076
C09759=1032.313,90.830,402.850,168.884,43.087,158.076
C09760=1032.307,90.581,402.869,168.881,43.088,158.076
C09761=1032.301,90.332,402.888,168.879,43.089,158.076
C09762=1032.295,90.083,402.907,168.877,43.091,158.076
C09763=1032.289,89.833,402.926,168.875,43.092,158.077
C09764=1032.283,89.584,402.945,168.872,43.093,158.077
C09765=1032.276,89.335,402.963,168.870,43.095,158.077
C09766=1032.270,89.086,402.982,168.867,43.096,158.077
C09767=1032.263,88.837,403.001,168.866,43.097,158.077
C09768=1032.257,88.588,403.019,168.863,43.099,158.077
C09769=1032.251,88.338,403.039,168.860,43.100,158.077
C09770=1032.245,88.089,403.056,168.859,43.102,158.077
C09771=1032.239,87.839,403.075,168.856,43.103,158.077
C09772=1032.232,87.590,403.094,168.854,43.104,158.077
C09773=1032.226,87.341,403.112,168.851,43.106,158.077
C09774=1032.219,87.092,403.131,168.849,43.107,158.077
C09775=1032.214,86.843,403.150,168.847,43.108,158.077
C09776=1032.207,86.594,403.169,168.845,43.110,158.078
C09777=1032.201,86.344,403.188,168.842,43.111,158.078
C09778=1032.195,86.095,403.206,168.839,43.113,158.078
C09779=1032.189,85.846,403.224,168.838,43.114,158.078
C09780=1032.183,85.597,403.242,168.835,43.115,158.078
C09781=1032.176,85.348,403.261,168.833,43.116,158.078
C09782=1032.170,85.099,403.280,168.830,43.118,158.078
C09783=1032.164,84.849,403.298,168.828,43.119,158.078
C09784=1032.158,84.600,403.317,168.826,43.120,158.078
C09785=1032.151,84.351,403.336,168.824,43.121,158.078
C09786=1032.145,84.101,403.354,168.821,43.123,158.078
C09787=1032.139,83.852,403.373,168.819,43.124,158.078
C09788=1032.133,83.603,403.391,168.817,43.125,158.078
C09789=1032.127,83.353,403.410,168.814,43.126,158.078
C09790=1032.121,83.105,403.428,168.812,43.128,158.079
C09791=1032.115,82.856,403.447,168.809,43.129,158.079
C09792=1032.108,82.606,403.465,168.808,43.130,158.079
C09793=1032.102,82.357,403.484,168.805,43.132,158.079
C09794=1032.096,82.108,403.502,168.803,43.133,158.079
C09795=1032.089,81.858,403.520,168.800,43.134,158.079
C09796=1032.083,81.609,403.539,168.799,43.136,158.079
C09797=1032.078,81.360,403.558,168.796,43.137,158.079
C09798=1032.072,81.111,403.576,168.794,43.138,158.079
C09799=1032.065,80.861,403.594,168.791,43.139,158.079
C09800=1032.059,80.612,403.613,168.790,43.141,158.079
C09801=1032.053,80.363,403.632,168.787,43.142,158.079
C09802=1032.046,80.113,403.650,168.785,43.143,158.079
C09803=1032.041,79.865,403.668,168.782,43.145,158.080
C09804=1032.034,79.616,403.686,168.779,43.146,158.080
C09805=1032.029,79.366,403.705,168.778,43.147,158.080
C09806=1032.022,79.116,403.724,168.775,43.148,158.080
C09807=1032.016,78.867,403.742,168.773,43.150,158.080
C09808=1032.010,78.618,403.760,168.770,43.151,158.080
C09809=1032.004,78.369,403.778,168.768,43.152,158.080
C09810=1031.998,78.119,403.796,168.766,43.154,158.080
C09811=1031.991,77.870,403.815,168.764,43.155,158.080
C09812=1031.985,77.621,403.833,168.761,43.156,158.080
C09813=1031.979,77.371,403.852,168.760,43.158,158.080
C09814=1031.973,77.123,403.870,168.757,43.159,158.080
C09815=1031.967,76.873,403.888,168.755,43.160,158.080
C09816=1031.960,76.588,403.909,168.752,43.162,158.080
C09817=1031.953,76.302,403.930,168.749,43.163,158.080
C09818=1031.945,76.016,403.951,168.747,43.165,158.081
C09819=1031.938,75.730,403.971,168.744,43.167,158.081
C09820=1031.932,75.481,403.989,168.741,43.168,158.081
C09821=1031.926,75.232,404.007,168.739,43.169,158.081
C09822=1031.920,74.983,404.026,168.737,43.171,158.081
C09823=1031.913,74.734,404.043,168.735,43.172,158.081
C09824=1031.907,74.485,404.062,168.732,43.173,158.081
C09825=1031.901,74.235,404.080,168.731,43.174,158.081
C09826=1031.895,73.986,404.098,168.728,43.176,158.081
C09827=1031.889,73.737,404.116,168.726,43.177,158.081
C09828=1031.883,73.487,404.134,168.723,43.178,158.081
C09829=1031.875,73.238,404.152,168.722,43.180,158.082
C09830=1031.870,72.989,404.169,168.719,43.181,158.082
C09831=1031.863,72.740,404.188,168.716,43.183,158.082
C09832=1031.857,72.490,404.206,168.714,43.184,158.082
C09833=1031.851,72.240,404.224,168.711,43.185,158.082
C09834=1031.845,71.992,404.242,168.710,43.186,158.082
C09835=1031.838,71.743,404.259,168.707,43.188,158.082
C09836=1031.832,71.493,404.277,168.705,43.189,158.082
C09837=1031.826,71.244,404.296,168.702,43.190,158.082
C09838=1031.820,70.995,404.314,168.701,43.192,158.082
C09839=1031.814,70.745,404.332,168.698,43.193,158.082
C09840=1031.807,70.496,404.350,168.696,43.195,158.082
C09841=1031.802,70.247,404.367,168.693,43.196,158.082
C09842=1031.795,69.997,404.385,168.692,43.197,158.082
C09843=1031.789,69.748,404.404,168.689,43.199,158.083
C09844=1031.783,69.499,404.422,168.686,43.200,158.083
C09845=1031.777,69.250,404.439,168.684,43.201,158.083
C09846=1031.771,69.000,404.457,168.682,43.203,158.083
C09847=1031.764,68.751,404.475,168.680,43.204,158.083
C09848=1031.759,68.502,404.493,168.677,43.206,158.083
C09849=1031.752,68.252,404.510,168.675,43.207,158.083
C09850=1031.746,68.003,404.528,168.673,43.208,158.083
C09851=1031.740,67.754,404.546,168.671,43.210,158.083
C09852=1031.733,67.505,404.564,168.668,43.211,158.083
C09853=1031.727,67.255,404.582,168.665,43.213,158.083
C09854=1031.721,67.006,404.599,168.664,43.214,158.083
C09855=1031.714,66.757,404.617,168.661,43.215,158.083
C09856=1031.708,66.507,404.634,168.659,43.216,158.084
C09857=1031.702,66.259,404.652,168.656,43.218,158.084
C09858=1031.696,66.009,404.670,168.655,43.219,158.084
C09859=1031.690,65.759,404.688,168.652,43.220,158.084
C09860=1031.683,65.511,404.705,168.650,43.221,158.084
C09861=1031.677,65.261,404.723,168.647,43.223,158.084
C09862=1031.670,65.011,404.740,168.646,43.224,158.084
C09863=1031.665,64.762,404.758,168.643,43.226,158.084
C09864=1031.659,64.513,404.776,168.640,43.227,158.084
C09865=1031.652,64.263,404.793,168.638,43.229,158.084
C09866=1031.646,64.015,404.811,168.636,43.230,158.084
C09867=1031.639,63.765,404.829,168.634,43.231,158.084
C09868=1031.634,63.516,404.846,168.631,43.233,158.085
C09869=1031.627,63.267,404.864,168.629,43.234,158.085
C09870=1031.621,63.017,404.882,168.627,43.236,158.085
C09871=1031.614,62.768,404.899,168.624,43.237,158.085
C09872=1031.608,62.519,404.916,168.622,43.239,158.085
C09873=1031.602,62.269,404.933,168.620,43.241,158.085
C09874=1031.595,62.020,404.950,168.618,43.242,158.085
C09875=1031.589,61.770,404.967,168.615,43.243,158.085
C09876=1031.582,61.521,404.985,168.612,43.245,158.085
C09877=1031.576,61.272,405.002,168.611,43.246,158.085
C09878=1031.569,61.023,405.020,168.608,43.247,158.085
C09879=1031.563,60.773,405.038,168.606,43.249,158.086
C09880=1031.556,60.487,405.057,168.604,43.251,158.086
C09881=1031.549,60.201,405.077,168.601,43.252,158.086
C09882=1031.542,59.915,405.097,168.598,43.254,158.086
C09883=1031.534,59.630,405.117,168.595,43.256,158.086
C09884=1031.528,59.381,405.133,168.593,43.257,158.086
C09885=1031.522,59.131,405.151,168.590,43.259,158.086
C09886=1031.515,58.883,405.168,168.588,43.260,158.086
C09887=1031.508,58.633,405.185,168.586,43.262,158.086
C09888=1031.502,58.383,405.203,168.584,43.263,158.086
C09889=1031.496,58.135,405.220,168.581,43.264,158.087
C09890=1031.489,57.885,405.237,168.579,43.266,158.087
C09891=1031.484,57.636,405.255,168.577,43.267,158.087
C09892=1031.477,57.386,405.272,168.574,43.269,158.087
C09893=1031.471,57.137,405.289,168.572,43.270,158.087
C09894=1031.464,56.888,405.306,168.569,43.271,158.087
C09895=1031.458,56.639,405.324,168.568,43.273,158.087
C09896=1031.452,56.389,405.340,168.565,43.274,158.087
C09897=1031.445,56.139,405.358,168.562,43.276,158.087
C09898=1031.440,55.890,405.375,168.560,43.277,158.087
C09899=1031.433,55.641,405.393,168.558,43.279,158.087
C09900=1031.427,55.392,405.409,168.556,43.280,158.088
C09901=1031.420,55.142,405.426,168.553,43.282,158.088
C09902=1031.414,54.893,405.444,168.551,43.283,158.088
C09903=1031.407,54.644,405.461,168.549,43.285,158.088
C09904=1031.402,54.394,405.477,168.546,43.286,158.088
C09905=1031.395,54.145,405.495,168.544,43.287,158.088
C09906=1031.389,53.896,405.512,168.542,43.289,158.088
C09907=1031.382,53.646,405.530,168.540,43.290,158.088
C09908=1031.376,53.397,405.546,168.537,43.292,158.088
C09909=1031.370,53.147,405.564,168.535,43.293,158.088
C09910=1031.364,52.899,405.581,168.533,43.294,158.088
C09911=1031.357,52.649,405.597,168.530,43.296,158.088
C09912=1031.352,52.400,405.615,168.528,43.297,158.089
C09913=1031.346,52.151,405.632,168.525,43.298,158.089
C09914=1031.339,51.901,405.649,168.524,43.300,158.089
C09915=1031.333,51.652,405.666,168.521,43.301,158.089
C09916=1031.327,51.402,405.683,168.519,43.302,158.089
C09917=1031.321,51.153,405.700,168.516,43.304,158.089
C09918=1031.314,50.904,405.717,168.514,43.305,158.089
C09919=1031.308,50.655,405.734,168.512,43.307,158.089
C09920=1031.302,50.405,405.751,168.509,43.308,158.089
C09921=1031.296,50.156,405.768,168.507,43.309,158.089
C09922=1031.290,49.906,405.784,168.505,43.311,158.089
C09923=1031.284,49.657,405.802,168.503,43.312,158.089
C09924=1031.277,49.408,405.819,168.500,43.314,158.090
C09925=1031.271,49.158,405.836,168.497,43.315,158.090
C09926=1031.264,48.909,405.853,168.496,43.316,158.090
C09927=1031.259,48.659,405.870,168.493,43.318,158.090
C09928=1031.252,48.410,405.887,168.491,43.319,158.090
C09929=1031.246,48.161,405.904,168.488,43.321,158.090
C09930=1031.240,47.912,405.920,168.487,43.322,158.090
C09931=1031.234,47.662,405.938,168.484,43.323,158.090
C09932=1031.228,47.413,405.955,168.482,43.325,158.090
C09933=1031.221,47.163,405.972,168.479,43.326,158.090
C09934=1031.215,46.914,405.988,168.476,43.327,158.090
C09935=1031.210,46.665,406.006,168.475,43.329,158.090
C09936=1031.203,46.415,406.022,168.472,43.330,158.090
C09937=1031.197,46.166,406.039,168.470,43.332,158.090
C09938=1031.191,45.917,406.056,168.468,43.333,158.090
C09939=1031.184,45.668,406.073,168.466,43.334,158.091
C09940=1031.179,45.418,406.090,168.463,43.336,158.091
C09941=1031.173,45.169,406.107,168.461,43.337,158.091
C09942=1031.166,44.919,406.123,168.458,43.338,158.091
C09943=1031.160,44.670,406.140,168.456,43.340,158.091
C09944=1031.153,44.384,406.160,168.454,43.341,158.091
C09945=1031.146,44.098,406.180,168.451,43.343,158.091
C09946=1031.139,43.812,406.198,168.449,43.344,158.091
C09947=1031.132,43.526,406.218,168.446,43.346,158.091
C09948=1031.126,43.276,406.234,168.443,43.347,158.091
C09949=1031.120,43.027,406.251,168.441,43.348,158.091
C09950=1031.114,42.778,406.268,168.439,43.350,158.091
C09951=1031.107,42.528,406.284,168.436,43.351,158.091
C09952=1031.101,42.279,406.300,168.434,43.352,158.092
C09953=1031.095,42.030,406.317,168.431,43.354,158.092
C09954=1031.088,41.780,406.334,168.430,43.355,158.092
C09955=1031.082,41.531,406.350,168.427,43.357,158.092
C09956=1031.076,41.282,406.367,168.424,43.358,158.092
C09957=1031.070,41.032,406.384,168.422,43.359,158.092
C09958=1031.064,40.783,406.400,168.420,43.361,158.092
C09959=1031.058,40.533,406.416,168.418,43.362,158.092
C09960=1031.051,40.284,406.434,168.415,43.364,158.092
C09961=1031.045,40.034,406.450,168.412,43.365,158.092
C09962=1031.039,39.785,406.466,168.411,43.366,158.092
C09963=1031.033,39.536,406.483,168.408,43.368,158.092
C09964=1031.026,39.286,406.500,168.406,43.369,158.092
C09965=1031.020,39.037,406.516,168.404,43.371,158.093
C09966=1031.014,38.788,406.532,168.401,43.372,158.093
C09967=1031.008,38.538,406.549,168.399,43.374,158.093
C09968=1031.001,38.289,406.566,168.396,43.375,158.093
C09969=1030.996,38.040,406.582,168.395,43.377,158.093
C09970=1030.990,37.790,406.598,168.392,43.378,158.093
C09971=1030.984,37.541,406.615,168.390,43.379,158.093
C09972=1030.977,37.291,406.631,168.387,43.381,158.093
C09973=1030.971,37.041,406.648,168.384,43.382,158.093
C09974=1030.964,36.792,406.663,168.383,43.384,158.093
C09975=1030.958,36.544,406.680,168.380,43.385,158.093
C09976=1030.952,36.294,406.697,168.377,43.387,158.093
C09977=1030.945,36.045,406.713,168.376,43.388,158.093
C09978=1030.939,35.795,406.729,168.373,43.390,158.094
C09979=1030.933,35.546,406.745,168.370,43.391,158.094
C09980=1030.926,35.296,406.762,168.368,43.392,158.094
C09981=1030.920,35.047,406.777,168.366,43.394,158.094
C09982=1030.914,34.797,406.794,168.364,43.395,158.094
C09983=1030.908,34.548,406.810,168.361,43.397,158.094
C09984=1030.901,34.298,406.826,168.359,43.398,158.094
C09985=1030.895,34.049,406.842,168.357,43.400,158.094
C09986=1030.889,33.800,406.858,168.354,43.401,158.094
C09987=1030.883,33.550,406.875,168.351,43.403,158.094
C09988=1030.876,33.301,406.890,168.350,43.404,158.094
C09989=1030.869,33.051,406.907,168.347,43.406,158.095
C09990=1030.864,32.802,406.923,168.344,43.407,158.095
C09991=1030.858,32.553,406.939,168.343,43.409,158.095
C09992=1030.851,32.303,406.955,168.340,43.410,158.095
C09993=1030.845,32.054,406.971,168.338,43.412,158.095
C09994=1030.839,31.805,406.988,168.335,43.413,158.095
C09995=1030.832,31.555,407.004,168.333,43.415,158.095
C09996=1030.826,31.306,407.020,168.331,43.416,158.095
//INST
///DATE 2021/06/25 14:48
///ATTR SC,RW,RJ
////FRAME ROBOT
///GROUP1 RB1
NOP
MOVL C00000 V=800.0 PL=0
MOVL C00001 V=800.0 PL=0
MOVL C00002 V=800.0 PL=0
MOVL C00003 V=800.0 PL=0
MOVL C00004 V=800.0 PL=0
MOVL C00005 V=800.0 PL=0
MOVL C00006 V=800.0 PL=0
MOVL C00007 V=800.0 PL=0
MOVL C00008 V=800.0 PL=0
MOVL C00009 V=800.0 PL=0
MOVL C00010 V=800.0 PL=0
MOVL C00011 V=800.0 PL=0
MOVL C00012 V=800.0 PL=0
MOVL C00013 V=800.0 PL=0
MOVL C00014 V=800.0 PL=0
MOVL C00015 V=800.0 PL=0
MOVL C00016 V=800.0 PL=0
MOVL C00017 V=800.0 PL=0
MOVL C00018 V=800.0 PL=0
MOVL C00019 V=800.0 PL=0
MOVL C00020 V=800.0 PL=0
MOVL C00021 V=800.0 PL=0
MOVL C00022 V=800.0 PL=0
MOVL C00023 V=800.0 PL=0
MOVL C00024 V=800.0 PL=0
MOVL C00025 V=800.0 PL=0
MOVL C00026 V=800.0 PL=0
MOVL C00027 V=800.0 PL=0
MOVL C00028 V=800.0 PL=0
MOVL C00029 V=800.0 PL=0
MOVL C00030 V=800.0 PL=0
MOVL C00031 V=800.0 PL=0
MOVL C00032 V=800.0 PL=0
MOVL C00033 V=800.0 PL=0
MOVL C00034 V=800.0 PL=0
MOVL C00035 V=800.0 PL=0
MOVL C00036 V=800.0 PL=0
MOVL C00037 V=800.0 PL=0
MOVL C00038 V=800.0 PL=0
MOVL C00039 V=800.0 PL=0
MOVL C00040 V=800.0 PL=0
MOVL C00041 V=800.0 PL=0
MOVL C00042 V=800.0 PL=0
MOVL C00043 V=800.0 PL=0
MOVL C00044 V=800.0 PL=0
MOVL C00045 V=800.0 PL=0
MOVL C00046 V=800.0 PL=0
MOVL C00047 V=800.0 PL=0
MOVL C00048 V=800.0 PL=0
MOVL C00049 V=800.0 PL=0
MOVL C00050 V=800.0 PL=0
MOVL C00051 V=800.0 PL=0
MOVL C00052 V=800.0 PL=0
MOVL C00053 V=800.0 PL=0
MOVL C00054 V=800.0 PL=0
MOVL C00055 V=800.0 PL=0
MOVL C00056 V=800.0 PL=0
MOVL C00057 V=800.0 PL=0
MOVL C00058 V=800.0 PL=0
MOVL C00059 V=800.0 PL=0
MOVL C00060 V=800.0 PL=0
MOVL C00061 V=800.0 PL=0
MOVL C00062 V=800.0 PL=0
MOVL C00063 V=800.0 PL=0
MOVL C00064 V=800.0 PL=0
MOVL C00065 V=800.0 PL=0
MOVL C00066 V=800.0 PL=0
MOVL C00067 V=800.0 PL=0
MOVL C00068 V=800.0 PL=0
MOVL C00069 V=800.0 PL=0
MOVL C00070 V=800.0 PL=0
MOVL C00071 V=800.0 PL=0
MOVL C00072 V=800.0 PL=0
MOVL C00073 V=800.0 PL=0
MOVL C00074 V=800.0 PL=0
MOVL C00075 V=800.0 PL=0
MOVL C00076 V=800.0 PL=0
MOVL C00077 V=800.0 PL=0
MOVL C00078 V=800.0 PL=0
MOVL C00079 V=800.0 PL=0
MOVL C00080 V=800.0 PL=0
MOVL C00081 V=800.0 PL=0
MOVL C00082 V=800.0 PL=0
MOVL C00083 V=800.0 PL=0
MOVL C00084 V=800.0 PL=0
MOVL C00085 V=800.0 PL=0
MOVL C00086 V=800.0 PL=0
MOVL C00087 V=800.0 PL=0
MOVL C00088 V=800.0 PL=0
MOVL C00089 V=800.0 PL=0
MOVL C00090 V=800.0 PL=0
MOVL C00091 V=800.0 PL=0
MOVL C00092 V=800.0 PL=0
MOVL C00093 V=800.0 PL=0
MOVL C00094 V=800.0 PL=0
MOVL C00095 V=800.0 PL=0
MOVL C00096 V=800.0 PL=0
MOVL C00097 V=800.0 PL=0
MOVL C00098 V=800.0 PL=0
MOVL C00099 V=800.0 PL=0
MOVL C00100 V=800.0 PL=0
MOVL C00101 V=800.0 PL=0
MOVL C00102 V=800.0 PL=0
MOVL C00103 V=800.0 PL=0
MOVL C00104 V=800.0 PL=0
MOVL C00105 V=800.0 PL=0
MOVL C00106 V=800.0 PL=0
MOVL C00107 V=800.0 PL=0
MOVL C00108 V=800.0 PL=0
MOVL C00109 V=800.0 PL=0
MOVL C00110 V=800.0 PL=0
MOVL C00111 V=800.0 PL=0
MOVL C00112 V=800.0 PL=0
MOVL C00113 V=800.0 PL=0
MOVL C00114 V=800.0 PL=0
MOVL C00115 V=800.0 PL=0
MOVL C00116 V=800.0 PL=0
MOVL C00117 V=800.0 PL=0
MOVL C00118 V=800.0 PL=0
MOVL C00119 V=800.0 PL=0
MOVL C00120 V=800.0 PL=0
MOVL C00121 V=800.0 PL=0
MOVL C00122 V=800.0 PL=0
MOVL C00123 V=800.0 PL=0
MOVL C00124 V=800.0 PL=0
MOVL C00125 V=800.0 PL=0
MOVL C00126 V=800.0 PL=0
MOVL C00127 V=800.0 PL=0
MOVL C00128 V=800.0 PL=0
MOVL C00129 V=800.0 PL=0
MOVL C00130 V=800.0 PL=0
MOVL C00131 V=800.0 PL=0
MOVL C00132 V=800.0 PL=0
MOVL C00133 V=800.0 PL=0
MOVL C00134 V=800.0 PL=0
MOVL C00135 V=800.0 PL=0
MOVL C00136 V=800.0 PL=0
MOVL C00137 V=800.0 PL=0
MOVL C00138 V=800.0 PL=0
MOVL C00139 V=800.0 PL=0
MOVL C00140 V=800.0 PL=0
MOVL C00141 V=800.0 PL=0
MOVL C00142 V=800.0 PL=0
MOVL C00143 V=800.0 PL=0
MOVL C00144 V=800.0 PL=0
MOVL C00145 V=800.0 PL=0
MOVL C00146 V=800.0 PL=0
MOVL C00147 V=800.0 PL=0
MOVL C00148 V=800.0 PL=0
MOVL C00149 V=800.0 PL=0
MOVL C00150 V=800.0 PL=0
MOVL C00151 V=800.0 PL=0
MOVL C00152 V=800.0 PL=0
MOVL C00153 V=800.0 PL=0
MOVL C00154 V=800.0 PL=0
MOVL C00155 V=800.0 PL=0
MOVL C00156 V=800.0 PL=0
MOVL C00157 V=800.0 PL=0
MOVL C00158 V=800.0 PL=0
MOVL C00159 V=800.0 PL=0
MOVL C00160 V=800.0 PL=0
MOVL C00161 V=800.0 PL=0
MOVL C00162 V=800.0 PL=0
MOVL C00163 V=800.0 PL=0
MOVL C00164 V=800.0 PL=0
MOVL C00165 V=800.0 PL=0
MOVL C00166 V=800.0 PL=0
MOVL C00167 V=800.0 PL=0
MOVL C00168 V=800.0 PL=0
MOVL C00169 V=800.0 PL=0
MOVL C00170 V=800.0 PL=0
MOVL C00171 V=800.0 PL=0
MOVL C00172 V=800.0 PL=0
MOVL C00173 V=800.0 PL=0
MOVL C00174 V=800.0 PL=0
MOVL C00175 V=800.0 PL=0
MOVL C00176 V=800.0 PL=0
MOVL C00177 V=800.0 PL=0
MOVL C00178 V=800.0 PL=0
MOVL C00179 V=800.0 PL=0
MOVL C00180 V=800.0 PL=0
MOVL C00181 V=800.0 PL=0
MOVL C00182 V=800.0 PL=0
MOVL C00183 V=800.0 PL=0
MOVL C00184 V=800.0 PL=0
MOVL C00185 V=800.0 PL=0
MOVL C00186 V=800.0 PL=0
MOVL C00187 V=800.0 PL=0
MOVL C00188 V=800.0 PL=0
MOVL C00189 V=800.0 PL=0
MOVL C00190 V=800.0 PL=0
MOVL C00191 V=800.0 PL=0
MOVL C00192 V=800.0 PL=0
MOVL C00193 V=800.0 PL=0
MOVL C00194 V=800.0 PL=0
MOVL C00195 V=800.0 PL=0
MOVL C00196 V=800.0 PL=0
MOVL C00197 V=800.0 PL=0
MOVL C00198 V=800.0 PL=0
MOVL C00199 V=800.0 PL=0
MOVL C00200 V=800.0 PL=0
MOVL C00201 V=800.0 PL=0
MOVL C00202 V=800.0 PL=0
MOVL C00203 V=800.0 PL=0
MOVL C00204 V=800.0 PL=0
MOVL C00205 V=800.0 PL=0
MOVL C00206 V=800.0 PL=0
MOVL C00207 V=800.0 PL=0
MOVL C00208 V=800.0 PL=0
MOVL C00209 V=800.0 PL=0
MOVL C00210 V=800.0 PL=0
MOVL C00211 V=800.0 PL=0
MOVL C00212 V=800.0 PL=0
MOVL C00213 V=800.0 PL=0
MOVL C00214 V=800.0 PL=0
MOVL C00215 V=800.0 PL=0
MOVL C00216 V=800.0 PL=0
MOVL C00217 V=800.0 PL=0
MOVL C00218 V=800.0 PL=0
MOVL C00219 V=800.0 PL=0
MOVL C00220 V=800.0 PL=0
MOVL C00221 V=800.0 PL=0
MOVL C00222 V=800.0 PL=0
MOVL C00223 V=800.0 PL=0
MOVL C00224 V=800.0 PL=0
MOVL C00225 V=800.0 PL=0
MOVL C00226 V=800.0 PL=0
MOVL C00227 V=800.0 PL=0
MOVL C00228 V=800.0 PL=0
MOVL C00229 V=800.0 PL=0
MOVL C00230 V=800.0 PL=0
MOVL C00231 V=800.0 PL=0
MOVL C00232 V=800.0 PL=0
MOVL C00233 V=800.0 PL=0
MOVL C00234 V=800.0 PL=0
MOVL C00235 V=800.0 PL=0
MOVL C00236 V=800.0 PL=0
MOVL C00237 V=800.0 PL=0
MOVL C00238 V=800.0 PL=0
MOVL C00239 V=800.0 PL=0
MOVL C00240 V=800.0 PL=0
MOVL C00241 V=800.0 PL=0
MOVL C00242 V=800.0 PL=0
MOVL C00243 V=800.0 PL=0
MOVL C00244 V=800.0 PL=0
MOVL C00245 V=800.0 PL=0
MOVL C00246 V=800.0 PL=0
MOVL C00247 V=800.0 PL=0
MOVL C00248 V=800.0 PL=0
MOVL C00249 V=800.0 PL=0
MOVL C00250 V=800.0 PL=0
MOVL C00251 V=800.0 PL=0
MOVL C00252 V=800.0 PL=0
MOVL C00253 V=800.0 PL=0
MOVL C00254 V=800.0 PL=0
MOVL C00255 V=800.0 PL=0
MOVL C00256 V=800.0 PL=0
MOVL C00257 V=800.0 PL=0
MOVL C00258 V=800.0 PL=0
MOVL C00259 V=800.0 PL=0
MOVL C00260 V=800.0 PL=0
MOVL C00261 V=800.0 PL=0
MOVL C00262 V=800.0 PL=0
MOVL C00263 V=800.0 PL=0
MOVL C00264 V=800.0 PL=0
MOVL C00265 V=800.0 PL=0
MOVL C00266 V=800.0 PL=0
MOVL C00267 V=800.0 PL=0
MOVL C00268 V=800.0 PL=0
MOVL C00269 V=800.0 PL=0
MOVL C00270 V=800.0 PL=0
MOVL C00271 V=800.0 PL=0
MOVL C00272 V=800.0 PL=0
MOVL C00273 V=800.0 PL=0
MOVL C00274 V=800.0 PL=0
MOVL C00275 V=800.0 PL=0
MOVL C00276 V=800.0 PL=0
MOVL C00277 V=800.0 PL=0
MOVL C00278 V=800.0 PL=0
MOVL C00279 V=800.0 PL=0
MOVL C00280 V=800.0 PL=0
MOVL C00281 V=800.0 PL=0
MOVL C00282 V=800.0 PL=0
MOVL C00283 V=800.0 PL=0
MOVL C00284 V=800.0 PL=0
MOVL C00285 V=800.0 PL=0
MOVL C00286 V=800.0 PL=0
MOVL C00287 V=800.0 PL=0
MOVL C00288 V=800.0 PL=0
MOVL C00289 V=800.0 PL=0
MOVL C00290 V=800.0 PL=0
MOVL C00291 V=800.0 PL=0
MOVL C00292 V=800.0 PL=0
MOVL C00293 V=800.0 PL=0
MOVL C00294 V=800.0 PL=0
MOVL C00295 V=800.0 PL=0
MOVL C00296 V=800.0 PL=0
MOVL C00297 V=800.0 PL=0
MOVL C00298 V=800.0 PL=0
MOVL C00299 V=800.0 PL=0
MOVL C00300 V=800.0 PL=0
MOVL C00301 V=800.0 PL=0
MOVL C00302 V=800.0 PL=0
MOVL C00303 V=800.0 PL=0
MOVL C00304 V=800.0 PL=0
MOVL C00305 V=800.0 PL=0
MOVL C00306 V=800.0 PL=0
MOVL C00307 V=800.0 PL=0
MOVL C00308 V=800.0 PL=0
MOVL C00309 V=800.0 PL=0
MOVL C00310 V=800.0 PL=0
MOVL C00311 V=800.0 PL=0
MOVL C00312 V=800.0 PL=0
MOVL C00313 V=800.0 PL=0
MOVL C00314 V=800.0 PL=0
MOVL C00315 V=800.0 PL=0
MOVL C00316 V=800.0 PL=0
MOVL C00317 V=800.0 PL=0
MOVL C00318 V=800.0 PL=0
MOVL C00319 V=800.0 PL=0
MOVL C00320 V=800.0 PL=0
MOVL C00321 V=800.0 PL=0
MOVL C00322 V=800.0 PL=0
MOVL C00323 V=800.0 PL=0
MOVL C00324 V=800.0 PL=0
MOVL C00325 V=800.0 PL=0
MOVL C00326 V=800.0 PL=0
MOVL C00327 V=800.0 PL=0
MOVL C00328 V=800.0 PL=0
MOVL C00329 V=800.0 PL=0
MOVL C00330 V=800.0 PL=0
MOVL C00331 V=800.0 PL=0
MOVL C00332 V=800.0 PL=0
MOVL C00333 V=800.0 PL=0
MOVL C00334 V=800.0 PL=0
MOVL C00335 V=800.0 PL=0
MOVL C00336 V=800.0 PL=0
MOVL C00337 V=800.0 PL=0
MOVL C00338 V=800.0 PL=0
MOVL C00339 V=800.0 PL=0
MOVL C00340 V=800.0 PL=0
MOVL C00341 V=800.0 PL=0
MOVL C00342 V=800.0 PL=0
MOVL C00343 V=800.0 PL=0
MOVL C00344 V=800.0 PL=0
MOVL C00345 V=800.0 PL=0
MOVL C00346 V=800.0 PL=0
MOVL C00347 V=800.0 PL=0
MOVL C00348 V=800.0 PL=0
MOVL C00349 V=800.0 PL=0
MOVL C00350 V=800.0 PL=0
MOVL C00351 V=800.0 PL=0
MOVL C00352 V=800.0 PL=0
MOVL C00353 V=800.0 PL=0
MOVL C00354 V=800.0 PL=0
MOVL C00355 V=800.0 PL=0
MOVL C00356 V=800.0 PL=0
MOVL C00357 V=800.0 PL=0
MOVL C00358 V=800.0 PL=0
MOVL C00359 V=800.0 PL=0
MOVL C00360 V=800.0 PL=0
MOVL C00361 V=800.0 PL=0
MOVL C00362 V=800.0 PL=0
MOVL C00363 V=800.0 PL=0
MOVL C00364 V=800.0 PL=0
MOVL C00365 V=800.0 PL=0
MOVL C00366 V=800.0 PL=0
MOVL C00367 V=800.0 PL=0
MOVL C00368 V=800.0 PL=0
MOVL C00369 V=800.0 PL=0
MOVL C00370 V=800.0 PL=0
MOVL C00371 V=800.0 PL=0
MOVL C00372 V=800.0 PL=0
MOVL C00373 V=800.0 PL=0
MOVL C00374 V=800.0 PL=0
MOVL C00375 V=800.0 PL=0
MOVL C00376 V=800.0 PL=0
MOVL C00377 V=800.0 PL=0
MOVL C00378 V=800.0 PL=0
MOVL C00379 V=800.0 PL=0
MOVL C00380 V=800.0 PL=0
MOVL C00381 V=800.0 PL=0
MOVL C00382 V=800.0 PL=0
MOVL C00383 V=800.0 PL=0
MOVL C00384 V=800.0 PL=0
MOVL C00385 V=800.0 PL=0
MOVL C00386 V=800.0 PL=0
MOVL C00387 V=800.0 PL=0
MOVL C00388 V=800.0 PL=0
MOVL C00389 V=800.0 PL=0
MOVL C00390 V=800.0 PL=0
MOVL C00391 V=800.0 PL=0
MOVL C00392 V=800.0 PL=0
MOVL C00393 V=800.0 PL=0
MOVL C00394 V=800.0 PL=0
MOVL C00395 V=800.0 PL=0
MOVL C00396 V=800.0 PL=0
MOVL C00397 V=800.0 PL=0
MOVL C00398 V=800.0 PL=0
MOVL C00399 V=800.0 PL=0
MOVL C00400 V=800.0 PL=0
MOVL C00401 V=800.0 PL=0
MOVL C00402 V=800.0 PL=0
MOVL C00403 V=800.0 PL=0
MOVL C00404 V=800.0 PL=0
MOVL C00405 V=800.0 PL=0
MOVL C00406 V=800.0 PL=0
MOVL C00407 V=800.0 PL=0
MOVL C00408 V=800.0 PL=0
MOVL C00409 V=800.0 PL=0
MOVL C00410 V=800.0 PL=0
MOVL C00411 V=800.0 PL=0
MOVL C00412 V=800.0 PL=0
MOVL C00413 V=800.0 PL=0
MOVL C00414 V=800.0 PL=0
MOVL C00415 V=800.0 PL=0
MOVL C00416 V=800.0 PL=0
MOVL C00417 V=800.0 PL=0
MOVL C00418 V=800.0 PL=0
MOVL C00419 V=800.0 PL=0
MOVL C00420 V=800.0 PL=0
MOVL C00421 V=800.0 PL=0
MOVL C00422 V=800.0 PL=0
MOVL C00423 V=800.0 PL=0
MOVL C00424 V=800.0 PL=0
MOVL C00425 V=800.0 PL=0
MOVL C00426 V=800.0 PL=0
MOVL C00427 V=800.0 PL=0
MOVL C00428 V=800.0 PL=0
MOVL C00429 V=800.0 PL=0
MOVL C00430 V=800.0 PL=0
MOVL C00431 V=800.0 PL=0
MOVL C00432 V=800.0 PL=0
MOVL C00433 V=800.0 PL=0
MOVL C00434 V=800.0 PL=0
MOVL C00435 V=800.0 PL=0
MOVL C00436 V=800.0 PL=0
MOVL C00437 V=800.0 PL=0
MOVL C00438 V=800.0 PL=0
MOVL C00439 V=800.0 PL=0
MOVL C00440 V=800.0 PL=0
MOVL C00441 V=800.0 PL=0
MOVL C00442 V=800.0 PL=0
MOVL C00443 V=800.0 PL=0
MOVL C00444 V=800.0 PL=0
MOVL C00445 V=800.0 PL=0
MOVL C00446 V=800.0 PL=0
MOVL C00447 V=800.0 PL=0
MOVL C00448 V=800.0 PL=0
MOVL C00449 V=800.0 PL=0
MOVL C00450 V=800.0 PL=0
MOVL C00451 V=800.0 PL=0
MOVL C00452 V=800.0 PL=0
MOVL C00453 V=800.0 PL=0
MOVL C00454 V=800.0 PL=0
MOVL C00455 V=800.0 PL=0
MOVL C00456 V=800.0 PL=0
MOVL C00457 V=800.0 PL=0
MOVL C00458 V=800.0 PL=0
MOVL C00459 V=800.0 PL=0
MOVL C00460 V=800.0 PL=0
MOVL C00461 V=800.0 PL=0
MOVL C00462 V=800.0 PL=0
MOVL C00463 V=800.0 PL=0
MOVL C00464 V=800.0 PL=0
MOVL C00465 V=800.0 PL=0
MOVL C00466 V=800.0 PL=0
MOVL C00467 V=800.0 PL=0
MOVL C00468 V=800.0 PL=0
MOVL C00469 V=800.0 PL=0
MOVL C00470 V=800.0 PL=0
MOVL C00471 V=800.0 PL=0
MOVL C00472 V=800.0 PL=0
MOVL C00473 V=800.0 PL=0
MOVL C00474 V=800.0 PL=0
MOVL C00475 V=800.0 PL=0
MOVL C00476 V=800.0 PL=0
MOVL C00477 V=800.0 PL=0
MOVL C00478 V=800.0 PL=0
MOVL C00479 V=800.0 PL=0
MOVL C00480 V=800.0 PL=0
MOVL C00481 V=800.0 PL=0
MOVL C00482 V=800.0 PL=0
MOVL C00483 V=800.0 PL=0
MOVL C00484 V=800.0 PL=0
MOVL C00485 V=800.0 PL=0
MOVL C00486 V=800.0 PL=0
MOVL C00487 V=800.0 PL=0
MOVL C00488 V=800.0 PL=0
MOVL C00489 V=800.0 PL=0
MOVL C00490 V=800.0 PL=0
MOVL C00491 V=800.0 PL=0
MOVL C00492 V=800.0 PL=0
MOVL C00493 V=800.0 PL=0
MOVL C00494 V=800.0 PL=0
MOVL C00495 V=800.0 PL=0
MOVL C00496 V=800.0 PL=0
MOVL C00497 V=800.0 PL=0
MOVL C00498 V=800.0 PL=0
MOVL C00499 V=800.0 PL=0
MOVL C00500 V=800.0 PL=0
MOVL C00501 V=800.0 PL=0
MOVL C00502 V=800.0 PL=0
MOVL C00503 V=800.0 PL=0
MOVL C00504 V=800.0 PL=0
MOVL C00505 V=800.0 PL=0
MOVL C00506 V=800.0 PL=0
MOVL C00507 V=800.0 PL=0
MOVL C00508 V=800.0 PL=0
MOVL C00509 V=800.0 PL=0
MOVL C00510 V=800.0 PL=0
MOVL C00511 V=800.0 PL=0
MOVL C00512 V=800.0 PL=0
MOVL C00513 V=800.0 PL=0
MOVL C00514 V=800.0 PL=0
MOVL C00515 V=800.0 PL=0
MOVL C00516 V=800.0 PL=0
MOVL C00517 V=800.0 PL=0
MOVL C00518 V=800.0 PL=0
MOVL C00519 V=800.0 PL=0
MOVL C00520 V=800.0 PL=0
MOVL C00521 V=800.0 PL=0
MOVL C00522 V=800.0 PL=0
MOVL C00523 V=800.0 PL=0
MOVL C00524 V=800.0 PL=0
MOVL C00525 V=800.0 PL=0
MOVL C00526 V=800.0 PL=0
MOVL C00527 V=800.0 PL=0
MOVL C00528 V=800.0 PL=0
MOVL C00529 V=800.0 PL=0
MOVL C00530 V=800.0 PL=0
MOVL C00531 V=800.0 PL=0
MOVL C00532 V=800.0 PL=0
MOVL C00533 V=800.0 PL=0
MOVL C00534 V=800.0 PL=0
MOVL C00535 V=800.0 PL=0
MOVL C00536 V=800.0 PL=0
MOVL C00537 V=800.0 PL=0
MOVL C00538 V=800.0 PL=0
MOVL C00539 V=800.0 PL=0
MOVL C00540 V=800.0 PL=0
MOVL C00541 V=800.0 PL=0
MOVL C00542 V=800.0 PL=0
MOVL C00543 V=800.0 PL=0
MOVL C00544 V=800.0 PL=0
MOVL C00545 V=800.0 PL=0
MOVL C00546 V=800.0 PL=0
MOVL C00547 V=800.0 PL=0
MOVL C00548 V=800.0 PL=0
MOVL C00549 V=800.0 PL=0
MOVL C00550 V=800.0 PL=0
MOVL C00551 V=800.0 PL=0
MOVL C00552 V=800.0 PL=0
MOVL C00553 V=800.0 PL=0
MOVL C00554 V=800.0 PL=0
MOVL C00555 V=800.0 PL=0
MOVL C00556 V=800.0 PL=0
MOVL C00557 V=800.0 PL=0
MOVL C00558 V=800.0 PL=0
MOVL C00559 V=800.0 PL=0
MOVL C00560 V=800.0 PL=0
MOVL C00561 V=800.0 PL=0
MOVL C00562 V=800.0 PL=0
MOVL C00563 V=800.0 PL=0
MOVL C00564 V=800.0 PL=0
MOVL C00565 V=800.0 PL=0
MOVL C00566 V=800.0 PL=0
MOVL C00567 V=800.0 PL=0
MOVL C00568 V=800.0 PL=0
MOVL C00569 V=800.0 PL=0
MOVL C00570 V=800.0 PL=0
MOVL C00571 V=800.0 PL=0
MOVL C00572 V=800.0 PL=0
MOVL C00573 V=800.0 PL=0
MOVL C00574 V=800.0 PL=0
MOVL C00575 V=800.0 PL=0
MOVL C00576 V=800.0 PL=0
MOVL C00577 V=800.0 PL=0
MOVL C00578 V=800.0 PL=0
MOVL C00579 V=800.0 PL=0
MOVL C00580 V=800.0 PL=0
MOVL C00581 V=800.0 PL=0
MOVL C00582 V=800.0 PL=0
MOVL C00583 V=800.0 PL=0
MOVL C00584 V=800.0 PL=0
MOVL C00585 V=800.0 PL=0
MOVL C00586 V=800.0 PL=0
MOVL C00587 V=800.0 PL=0
MOVL C00588 V=800.0 PL=0
MOVL C00589 V=800.0 PL=0
MOVL C00590 V=800.0 PL=0
MOVL C00591 V=800.0 PL=0
MOVL C00592 V=800.0 PL=0
MOVL C00593 V=800.0 PL=0
MOVL C00594 V=800.0 PL=0
MOVL C00595 V=800.0 PL=0
MOVL C00596 V=800.0 PL=0
MOVL C00597 V=800.0 PL=0
MOVL C00598 V=800.0 PL=0
MOVL C00599 V=800.0 PL=0
MOVL C00600 V=800.0 PL=0
MOVL C00601 V=800.0 PL=0
MOVL C00602 V=800.0 PL=0
MOVL C00603 V=800.0 PL=0
MOVL C00604 V=800.0 PL=0
MOVL C00605 V=800.0 PL=0
MOVL C00606 V=800.0 PL=0
MOVL C00607 V=800.0 PL=0
MOVL C00608 V=800.0 PL=0
MOVL C00609 V=800.0 PL=0
MOVL C00610 V=800.0 PL=0
MOVL C00611 V=800.0 PL=0
MOVL C00612 V=800.0 PL=0
MOVL C00613 V=800.0 PL=0
MOVL C00614 V=800.0 PL=0
MOVL C00615 V=800.0 PL=0
MOVL C00616 V=800.0 PL=0
MOVL C00617 V=800.0 PL=0
MOVL C00618 V=800.0 PL=0
MOVL C00619 V=800.0 PL=0
MOVL C00620 V=800.0 PL=0
MOVL C00621 V=800.0 PL=0
MOVL C00622 V=800.0 PL=0
MOVL C00623 V=800.0 PL=0
MOVL C00624 V=800.0 PL=0
MOVL C00625 V=800.0 PL=0
MOVL C00626 V=800.0 PL=0
MOVL C00627 V=800.0 PL=0
MOVL C00628 V=800.0 PL=0
MOVL C00629 V=800.0 PL=0
MOVL C00630 V=800.0 PL=0
MOVL C00631 V=800.0 PL=0
MOVL C00632 V=800.0 PL=0
MOVL C00633 V=800.0 PL=0
MOVL C00634 V=800.0 PL=0
MOVL C00635 V=800.0 PL=0
MOVL C00636 V=800.0 PL=0
MOVL C00637 V=800.0 PL=0
MOVL C00638 V=800.0 PL=0
MOVL C00639 V=800.0 PL=0
MOVL C00640 V=800.0 PL=0
MOVL C00641 V=800.0 PL=0
MOVL C00642 V=800.0 PL=0
MOVL C00643 V=800.0 PL=0
MOVL C00644 V=800.0 PL=0
MOVL C00645 V=800.0 PL=0
MOVL C00646 V=800.0 PL=0
MOVL C00647 V=800.0 PL=0
MOVL C00648 V=800.0 PL=0
MOVL C00649 V=800.0 PL=0
MOVL C00650 V=800.0 PL=0
MOVL C00651 V=800.0 PL=0
MOVL C00652 V=800.0 PL=0
MOVL C00653 V=800.0 PL=0
MOVL C00654 V=800.0 PL=0
MOVL C00655 V=800.0 PL=0
MOVL C00656 V=800.0 PL=0
MOVL C00657 V=800.0 PL=0
MOVL C00658 V=800.0 PL=0
MOVL C00659 V=800.0 PL=0
MOVL C00660 V=800.0 PL=0
MOVL C00661 V=800.0 PL=0
MOVL C00662 V=800.0 PL=0
MOVL C00663 V=800.0 PL=0
MOVL C00664 V=800.0 PL=0
MOVL C00665 V=800.0 PL=0
MOVL C00666 V=800.0 PL=0
MOVL C00667 V=800.0 PL=0
MOVL C00668 V=800.0 PL=0
MOVL C00669 V=800.0 PL=0
MOVL C00670 V=800.0 PL=0
MOVL C00671 V=800.0 PL=0
MOVL C00672 V=800.0 PL=0
MOVL C00673 V=800.0 PL=0
MOVL C00674 V=800.0 PL=0
MOVL C00675 V=800.0 PL=0
MOVL C00676 V=800.0 PL=0
MOVL C00677 V=800.0 PL=0
MOVL C00678 V=800.0 PL=0
MOVL C00679 V=800.0 PL=0
MOVL C00680 V=800.0 PL=0
MOVL C00681 V=800.0 PL=0
MOVL C00682 V=800.0 PL=0
MOVL C00683 V=800.0 PL=0
MOVL C00684 V=800.0 PL=0
MOVL C00685 V=800.0 PL=0
MOVL C00686 V=800.0 PL=0
MOVL C00687 V=800.0 PL=0
MOVL C00688 V=800.0 PL=0
MOVL C00689 V=800.0 PL=0
MOVL C00690 V=800.0 PL=0
MOVL C00691 V=800.0 PL=0
MOVL C00692 V=800.0 PL=0
MOVL C00693 V=800.0 PL=0
MOVL C00694 V=800.0 PL=0
MOVL C00695 V=800.0 PL=0
MOVL C00696 V=800.0 PL=0
MOVL C00697 V=800.0 PL=0
MOVL C00698 V=800.0 PL=0
MOVL C00699 V=800.0 PL=0
MOVL C00700 V=800.0 PL=0
MOVL C00701 V=800.0 PL=0
MOVL C00702 V=800.0 PL=0
MOVL C00703 V=800.0 PL=0
MOVL C00704 V=800.0 PL=0
MOVL C00705 V=800.0 PL=0
MOVL C00706 V=800.0 PL=0
MOVL C00707 V=800.0 PL=0
MOVL C00708 V=800.0 PL=0
MOVL C00709 V=800.0 PL=0
MOVL C00710 V=800.0 PL=0
MOVL C00711 V=800.0 PL=0
MOVL C00712 V=800.0 PL=0
MOVL C00713 V=800.0 PL=0
MOVL C00714 V=800.0 PL=0
MOVL C00715 V=800.0 PL=0
MOVL C00716 V=800.0 PL=0
MOVL C00717 V=800.0 PL=0
MOVL C00718 V=800.0 PL=0
MOVL C00719 V=800.0 PL=0
MOVL C00720 V=800.0 PL=0
MOVL C00721 V=800.0 PL=0
MOVL C00722 V=800.0 PL=0
MOVL C00723 V=800.0 PL=0
MOVL C00724 V=800.0 PL=0
MOVL C00725 V=800.0 PL=0
MOVL C00726 V=800.0 PL=0
MOVL C00727 V=800.0 PL=0
MOVL C00728 V=800.0 PL=0
MOVL C00729 V=800.0 PL=0
MOVL C00730 V=800.0 PL=0
MOVL C00731 V=800.0 PL=0
MOVL C00732 V=800.0 PL=0
MOVL C00733 V=800.0 PL=0
MOVL C00734 V=800.0 PL=0
MOVL C00735 V=800.0 PL=0
MOVL C00736 V=800.0 PL=0
MOVL C00737 V=800.0 PL=0
MOVL C00738 V=800.0 PL=0
MOVL C00739 V=800.0 PL=0
MOVL C00740 V=800.0 PL=0
MOVL C00741 V=800.0 PL=0
MOVL C00742 V=800.0 PL=0
MOVL C00743 V=800.0 PL=0
MOVL C00744 V=800.0 PL=0
MOVL C00745 V=800.0 PL=0
MOVL C00746 V=800.0 PL=0
MOVL C00747 V=800.0 PL=0
MOVL C00748 V=800.0 PL=0
MOVL C00749 V=800.0 PL=0
MOVL C00750 V=800.0 PL=0
MOVL C00751 V=800.0 PL=0
MOVL C00752 V=800.0 PL=0
MOVL C00753 V=800.0 PL=0
MOVL C00754 V=800.0 PL=0
MOVL C00755 V=800.0 PL=0
MOVL C00756 V=800.0 PL=0
MOVL C00757 V=800.0 PL=0
MOVL C00758 V=800.0 PL=0
MOVL C00759 V=800.0 PL=0
MOVL C00760 V=800.0 PL=0
MOVL C00761 V=800.0 PL=0
MOVL C00762 V=800.0 PL=0
MOVL C00763 V=800.0 PL=0
MOVL C00764 V=800.0 PL=0
MOVL C00765 V=800.0 PL=0
MOVL C00766 V=800.0 PL=0
MOVL C00767 V=800.0 PL=0
MOVL C00768 V=800.0 PL=0
MOVL C00769 V=800.0 PL=0
MOVL C00770 V=800.0 PL=0
MOVL C00771 V=800.0 PL=0
MOVL C00772 V=800.0 PL=0
MOVL C00773 V=800.0 PL=0
MOVL C00774 V=800.0 PL=0
MOVL C00775 V=800.0 PL=0
MOVL C00776 V=800.0 PL=0
MOVL C00777 V=800.0 PL=0
MOVL C00778 V=800.0 PL=0
MOVL C00779 V=800.0 PL=0
MOVL C00780 V=800.0 PL=0
MOVL C00781 V=800.0 PL=0
MOVL C00782 V=800.0 PL=0
MOVL C00783 V=800.0 PL=0
MOVL C00784 V=800.0 PL=0
MOVL C00785 V=800.0 PL=0
MOVL C00786 V=800.0 PL=0
MOVL C00787 V=800.0 PL=0
MOVL C00788 V=800.0 PL=0
MOVL C00789 V=800.0 PL=0
MOVL C00790 V=800.0 PL=0
MOVL C00791 V=800.0 PL=0
MOVL C00792 V=800.0 PL=0
MOVL C00793 V=800.0 PL=0
MOVL C00794 V=800.0 PL=0
MOVL C00795 V=800.0 PL=0
MOVL C00796 V=800.0 PL=0
MOVL C00797 V=800.0 PL=0
MOVL C00798 V=800.0 PL=0
MOVL C00799 V=800.0 PL=0
MOVL C00800 V=800.0 PL=0
MOVL C00801 V=800.0 PL=0
MOVL C00802 V=800.0 PL=0
MOVL C00803 V=800.0 PL=0
MOVL C00804 V=800.0 PL=0
MOVL C00805 V=800.0 PL=0
MOVL C00806 V=800.0 PL=0
MOVL C00807 V=800.0 PL=0
MOVL C00808 V=800.0 PL=0
MOVL C00809 V=800.0 PL=0
MOVL C00810 V=800.0 PL=0
MOVL C00811 V=800.0 PL=0
MOVL C00812 V=800.0 PL=0
MOVL C00813 V=800.0 PL=0
MOVL C00814 V=800.0 PL=0
MOVL C00815 V=800.0 PL=0
MOVL C00816 V=800.0 PL=0
MOVL C00817 V=800.0 PL=0
MOVL C00818 V=800.0 PL=0
MOVL C00819 V=800.0 PL=0
MOVL C00820 V=800.0 PL=0
MOVL C00821 V=800.0 PL=0
MOVL C00822 V=800.0 PL=0
MOVL C00823 V=800.0 PL=0
MOVL C00824 V=800.0 PL=0
MOVL C00825 V=800.0 PL=0
MOVL C00826 V=800.0 PL=0
MOVL C00827 V=800.0 PL=0
MOVL C00828 V=800.0 PL=0
MOVL C00829 V=800.0 PL=0
MOVL C00830 V=800.0 PL=0
MOVL C00831 V=800.0 PL=0
MOVL C00832 V=800.0 PL=0
MOVL C00833 V=800.0 PL=0
MOVL C00834 V=800.0 PL=0
MOVL C00835 V=800.0 PL=0
MOVL C00836 V=800.0 PL=0
MOVL C00837 V=800.0 PL=0
MOVL C00838 V=800.0 PL=0
MOVL C00839 V=800.0 PL=0
MOVL C00840 V=800.0 PL=0
MOVL C00841 V=800.0 PL=0
MOVL C00842 V=800.0 PL=0
MOVL C00843 V=800.0 PL=0
MOVL C00844 V=800.0 PL=0
MOVL C00845 V=800.0 PL=0
MOVL C00846 V=800.0 PL=0
MOVL C00847 V=800.0 PL=0
MOVL C00848 V=800.0 PL=0
MOVL C00849 V=800.0 PL=0
MOVL C00850 V=800.0 PL=0
MOVL C00851 V=800.0 PL=0
MOVL C00852 V=800.0 PL=0
MOVL C00853 V=800.0 PL=0
MOVL C00854 V=800.0 PL=0
MOVL C00855 V=800.0 PL=0
MOVL C00856 V=800.0 PL=0
MOVL C00857 V=800.0 PL=0
MOVL C00858 V=800.0 PL=0
MOVL C00859 V=800.0 PL=0
MOVL C00860 V=800.0 PL=0
MOVL C00861 V=800.0 PL=0
MOVL C00862 V=800.0 PL=0
MOVL C00863 V=800.0 PL=0
MOVL C00864 V=800.0 PL=0
MOVL C00865 V=800.0 PL=0
MOVL C00866 V=800.0 PL=0
MOVL C00867 V=800.0 PL=0
MOVL C00868 V=800.0 PL=0
MOVL C00869 V=800.0 PL=0
MOVL C00870 V=800.0 PL=0
MOVL C00871 V=800.0 PL=0
MOVL C00872 V=800.0 PL=0
MOVL C00873 V=800.0 PL=0
MOVL C00874 V=800.0 PL=0
MOVL C00875 V=800.0 PL=0
MOVL C00876 V=800.0 PL=0
MOVL C00877 V=800.0 PL=0
MOVL C00878 V=800.0 PL=0
MOVL C00879 V=800.0 PL=0
MOVL C00880 V=800.0 PL=0
MOVL C00881 V=800.0 PL=0
MOVL C00882 V=800.0 PL=0
MOVL C00883 V=800.0 PL=0
MOVL C00884 V=800.0 PL=0
MOVL C00885 V=800.0 PL=0
MOVL C00886 V=800.0 PL=0
MOVL C00887 V=800.0 PL=0
MOVL C00888 V=800.0 PL=0
MOVL C00889 V=800.0 PL=0
MOVL C00890 V=800.0 PL=0
MOVL C00891 V=800.0 PL=0
MOVL C00892 V=800.0 PL=0
MOVL C00893 V=800.0 PL=0
MOVL C00894 V=800.0 PL=0
MOVL C00895 V=800.0 PL=0
MOVL C00896 V=800.0 PL=0
MOVL C00897 V=800.0 PL=0
MOVL C00898 V=800.0 PL=0
MOVL C00899 V=800.0 PL=0
MOVL C00900 V=800.0 PL=0
MOVL C00901 V=800.0 PL=0
MOVL C00902 V=800.0 PL=0
MOVL C00903 V=800.0 PL=0
MOVL C00904 V=800.0 PL=0
MOVL C00905 V=800.0 PL=0
MOVL C00906 V=800.0 PL=0
MOVL C00907 V=800.0 PL=0
MOVL C00908 V=800.0 PL=0
MOVL C00909 V=800.0 PL=0
MOVL C00910 V=800.0 PL=0
MOVL C00911 V=800.0 PL=0
MOVL C00912 V=800.0 PL=0
MOVL C00913 V=800.0 PL=0
MOVL C00914 V=800.0 PL=0
MOVL C00915 V=800.0 PL=0
MOVL C00916 V=800.0 PL=0
MOVL C00917 V=800.0 PL=0
MOVL C00918 V=800.0 PL=0
MOVL C00919 V=800.0 PL=0
MOVL C00920 V=800.0 PL=0
MOVL C00921 V=800.0 PL=0
MOVL C00922 V=800.0 PL=0
MOVL C00923 V=800.0 PL=0
MOVL C00924 V=800.0 PL=0
MOVL C00925 V=800.0 PL=0
MOVL C00926 V=800.0 PL=0
MOVL C00927 V=800.0 PL=0
MOVL C00928 V=800.0 PL=0
MOVL C00929 V=800.0 PL=0
MOVL C00930 V=800.0 PL=0
MOVL C00931 V=800.0 PL=0
MOVL C00932 V=800.0 PL=0
MOVL C00933 V=800.0 PL=0
MOVL C00934 V=800.0 PL=0
MOVL C00935 V=800.0 PL=0
MOVL C00936 V=800.0 PL=0
MOVL C00937 V=800.0 PL=0
MOVL C00938 V=800.0 PL=0
MOVL C00939 V=800.0 PL=0
MOVL C00940 V=800.0 PL=0
MOVL C00941 V=800.0 PL=0
MOVL C00942 V=800.0 PL=0
MOVL C00943 V=800.0 PL=0
MOVL C00944 V=800.0 PL=0
MOVL C00945 V=800.0 PL=0
MOVL C00946 V=800.0 PL=0
MOVL C00947 V=800.0 PL=0
MOVL C00948 V=800.0 PL=0
MOVL C00949 V=800.0 PL=0
MOVL C00950 V=800.0 PL=0
MOVL C00951 V=800.0 PL=0
MOVL C00952 V=800.0 PL=0
MOVL C00953 V=800.0 PL=0
MOVL C00954 V=800.0 PL=0
MOVL C00955 V=800.0 PL=0
MOVL C00956 V=800.0 PL=0
MOVL C00957 V=800.0 PL=0
MOVL C00958 V=800.0 PL=0
MOVL C00959 V=800.0 PL=0
MOVL C00960 V=800.0 PL=0
MOVL C00961 V=800.0 PL=0
MOVL C00962 V=800.0 PL=0
MOVL C00963 V=800.0 PL=0
MOVL C00964 V=800.0 PL=0
MOVL C00965 V=800.0 PL=0
MOVL C00966 V=800.0 PL=0
MOVL C00967 V=800.0 PL=0
MOVL C00968 V=800.0 PL=0
MOVL C00969 V=800.0 PL=0
MOVL C00970 V=800.0 PL=0
MOVL C00971 V=800.0 PL=0
MOVL C00972 V=800.0 PL=0
MOVL C00973 V=800.0 PL=0
MOVL C00974 V=800.0 PL=0
MOVL C00975 V=800.0 PL=0
MOVL C00976 V=800.0 PL=0
MOVL C00977 V=800.0 PL=0
MOVL C00978 V=800.0 PL=0
MOVL C00979 V=800.0 PL=0
MOVL C00980 V=800.0 PL=0
MOVL C00981 V=800.0 PL=0
MOVL C00982 V=800.0 PL=0
MOVL C00983 V=800.0 PL=0
MOVL C00984 V=800.0 PL=0
MOVL C00985 V=800.0 PL=0
MOVL C00986 V=800.0 PL=0
MOVL C00987 V=800.0 PL=0
MOVL C00988 V=800.0 PL=0
MOVL C00989 V=800.0 PL=0
MOVL C00990 V=800.0 PL=0
MOVL C00991 V=800.0 PL=0
MOVL C00992 V=800.0 PL=0
MOVL C00993 V=800.0 PL=0
MOVL C00994 V=800.0 PL=0
MOVL C00995 V=800.0 PL=0
MOVL C00996 V=800.0 PL=0
MOVL C00997 V=800.0 PL=0
MOVL C00998 V=800.0 PL=0
MOVL C00999 V=800.0 PL=0
MOVL C01000 V=800.0 PL=0
MOVL C01001 V=800.0 PL=0
MOVL C01002 V=800.0 PL=0
MOVL C01003 V=800.0 PL=0
MOVL C01004 V=800.0 PL=0
MOVL C01005 V=800.0 PL=0
MOVL C01006 V=800.0 PL=0
MOVL C01007 V=800.0 PL=0
MOVL C01008 V=800.0 PL=0
MOVL C01009 V=800.0 PL=0
MOVL C01010 V=800.0 PL=0
MOVL C01011 V=800.0 PL=0
MOVL C01012 V=800.0 PL=0
MOVL C01013 V=800.0 PL=0
MOVL C01014 V=800.0 PL=0
MOVL C01015 V=800.0 PL=0
MOVL C01016 V=800.0 PL=0
MOVL C01017 V=800.0 PL=0
MOVL C01018 V=800.0 PL=0
MOVL C01019 V=800.0 PL=0
MOVL C01020 V=800.0 PL=0
MOVL C01021 V=800.0 PL=0
MOVL C01022 V=800.0 PL=0
MOVL C01023 V=800.0 PL=0
MOVL C01024 V=800.0 PL=0
MOVL C01025 V=800.0 PL=0
MOVL C01026 V=800.0 PL=0
MOVL C01027 V=800.0 PL=0
MOVL C01028 V=800.0 PL=0
MOVL C01029 V=800.0 PL=0
MOVL C01030 V=800.0 PL=0
MOVL C01031 V=800.0 PL=0
MOVL C01032 V=800.0 PL=0
MOVL C01033 V=800.0 PL=0
MOVL C01034 V=800.0 PL=0
MOVL C01035 V=800.0 PL=0
MOVL C01036 V=800.0 PL=0
MOVL C01037 V=800.0 PL=0
MOVL C01038 V=800.0 PL=0
MOVL C01039 V=800.0 PL=0
MOVL C01040 V=800.0 PL=0
MOVL C01041 V=800.0 PL=0
MOVL C01042 V=800.0 PL=0
MOVL C01043 V=800.0 PL=0
MOVL C01044 V=800.0 PL=0
MOVL C01045 V=800.0 PL=0
MOVL C01046 V=800.0 PL=0
MOVL C01047 V=800.0 PL=0
MOVL C01048 V=800.0 PL=0
MOVL C01049 V=800.0 PL=0
MOVL C01050 V=800.0 PL=0
MOVL C01051 V=800.0 PL=0
MOVL C01052 V=800.0 PL=0
MOVL C01053 V=800.0 PL=0
MOVL C01054 V=800.0 PL=0
MOVL C01055 V=800.0 PL=0
MOVL C01056 V=800.0 PL=0
MOVL C01057 V=800.0 PL=0
MOVL C01058 V=800.0 PL=0
MOVL C01059 V=800.0 PL=0
MOVL C01060 V=800.0 PL=0
MOVL C01061 V=800.0 PL=0
MOVL C01062 V=800.0 PL=0
MOVL C01063 V=800.0 PL=0
MOVL C01064 V=800.0 PL=0
MOVL C01065 V=800.0 PL=0
MOVL C01066 V=800.0 PL=0
MOVL C01067 V=800.0 PL=0
MOVL C01068 V=800.0 PL=0
MOVL C01069 V=800.0 PL=0
MOVL C01070 V=800.0 PL=0
MOVL C01071 V=800.0 PL=0
MOVL C01072 V=800.0 PL=0
MOVL C01073 V=800.0 PL=0
MOVL C01074 V=800.0 PL=0
MOVL C01075 V=800.0 PL=0
MOVL C01076 V=800.0 PL=0
MOVL C01077 V=800.0 PL=0
MOVL C01078 V=800.0 PL=0
MOVL C01079 V=800.0 PL=0
MOVL C01080 V=800.0 PL=0
MOVL C01081 V=800.0 PL=0
MOVL C01082 V=800.0 PL=0
MOVL C01083 V=800.0 PL=0
MOVL C01084 V=800.0 PL=0
MOVL C01085 V=800.0 PL=0
MOVL C01086 V=800.0 PL=0
MOVL C01087 V=800.0 PL=0
MOVL C01088 V=800.0 PL=0
MOVL C01089 V=800.0 PL=0
MOVL C01090 V=800.0 PL=0
MOVL C01091 V=800.0 PL=0
MOVL C01092 V=800.0 PL=0
MOVL C01093 V=800.0 PL=0
MOVL C01094 V=800.0 PL=0
MOVL C01095 V=800.0 PL=0
MOVL C01096 V=800.0 PL=0
MOVL C01097 V=800.0 PL=0
MOVL C01098 V=800.0 PL=0
MOVL C01099 V=800.0 PL=0
MOVL C01100 V=800.0 PL=0
MOVL C01101 V=800.0 PL=0
MOVL C01102 V=800.0 PL=0
MOVL C01103 V=800.0 PL=0
MOVL C01104 V=800.0 PL=0
MOVL C01105 V=800.0 PL=0
MOVL C01106 V=800.0 PL=0
MOVL C01107 V=800.0 PL=0
MOVL C01108 V=800.0 PL=0
MOVL C01109 V=800.0 PL=0
MOVL C01110 V=800.0 PL=0
MOVL C01111 V=800.0 PL=0
MOVL C01112 V=800.0 PL=0
MOVL C01113 V=800.0 PL=0
MOVL C01114 V=800.0 PL=0
MOVL C01115 V=800.0 PL=0
MOVL C01116 V=800.0 PL=0
MOVL C01117 V=800.0 PL=0
MOVL C01118 V=800.0 PL=0
MOVL C01119 V=800.0 PL=0
MOVL C01120 V=800.0 PL=0
MOVL C01121 V=800.0 PL=0
MOVL C01122 V=800.0 PL=0
MOVL C01123 V=800.0 PL=0
MOVL C01124 V=800.0 PL=0
MOVL C01125 V=800.0 PL=0
MOVL C01126 V=800.0 PL=0
MOVL C01127 V=800.0 PL=0
MOVL C01128 V=800.0 PL=0
MOVL C01129 V=800.0 PL=0
MOVL C01130 V=800.0 PL=0
MOVL C01131 V=800.0 PL=0
MOVL C01132 V=800.0 PL=0
MOVL C01133 V=800.0 PL=0
MOVL C01134 V=800.0 PL=0
MOVL C01135 V=800.0 PL=0
MOVL C01136 V=800.0 PL=0
MOVL C01137 V=800.0 PL=0
MOVL C01138 V=800.0 PL=0
MOVL C01139 V=800.0 PL=0
MOVL C01140 V=800.0 PL=0
MOVL C01141 V=800.0 PL=0
MOVL C01142 V=800.0 PL=0
MOVL C01143 V=800.0 PL=0
MOVL C01144 V=800.0 PL=0
MOVL C01145 V=800.0 PL=0
MOVL C01146 V=800.0 PL=0
MOVL C01147 V=800.0 PL=0
MOVL C01148 V=800.0 PL=0
MOVL C01149 V=800.0 PL=0
MOVL C01150 V=800.0 PL=0
MOVL C01151 V=800.0 PL=0
MOVL C01152 V=800.0 PL=0
MOVL C01153 V=800.0 PL=0
MOVL C01154 V=800.0 PL=0
MOVL C01155 V=800.0 PL=0
MOVL C01156 V=800.0 PL=0
MOVL C01157 V=800.0 PL=0
MOVL C01158 V=800.0 PL=0
MOVL C01159 V=800.0 PL=0
MOVL C01160 V=800.0 PL=0
MOVL C01161 V=800.0 PL=0
MOVL C01162 V=800.0 PL=0
MOVL C01163 V=800.0 PL=0
MOVL C01164 V=800.0 PL=0
MOVL C01165 V=800.0 PL=0
MOVL C01166 V=800.0 PL=0
MOVL C01167 V=800.0 PL=0
MOVL C01168 V=800.0 PL=0
MOVL C01169 V=800.0 PL=0
MOVL C01170 V=800.0 PL=0
MOVL C01171 V=800.0 PL=0
MOVL C01172 V=800.0 PL=0
MOVL C01173 V=800.0 PL=0
MOVL C01174 V=800.0 PL=0
MOVL C01175 V=800.0 PL=0
MOVL C01176 V=800.0 PL=0
MOVL C01177 V=800.0 PL=0
MOVL C01178 V=800.0 PL=0
MOVL C01179 V=800.0 PL=0
MOVL C01180 V=800.0 PL=0
MOVL C01181 V=800.0 PL=0
MOVL C01182 V=800.0 PL=0
MOVL C01183 V=800.0 PL=0
MOVL C01184 V=800.0 PL=0
MOVL C01185 V=800.0 PL=0
MOVL C01186 V=800.0 PL=0
MOVL C01187 V=800.0 PL=0
MOVL C01188 V=800.0 PL=0
MOVL C01189 V=800.0 PL=0
MOVL C01190 V=800.0 PL=0
MOVL C01191 V=800.0 PL=0
MOVL C01192 V=800.0 PL=0
MOVL C01193 V=800.0 PL=0
MOVL C01194 V=800.0 PL=0
MOVL C01195 V=800.0 PL=0
MOVL C01196 V=800.0 PL=0
MOVL C01197 V=800.0 PL=0
MOVL C01198 V=800.0 PL=0
MOVL C01199 V=800.0 PL=0
MOVL C01200 V=800.0 PL=0
MOVL C01201 V=800.0 PL=0
MOVL C01202 V=800.0 PL=0
MOVL C01203 V=800.0 PL=0
MOVL C01204 V=800.0 PL=0
MOVL C01205 V=800.0 PL=0
MOVL C01206 V=800.0 PL=0
MOVL C01207 V=800.0 PL=0
MOVL C01208 V=800.0 PL=0
MOVL C01209 V=800.0 PL=0
MOVL C01210 V=800.0 PL=0
MOVL C01211 V=800.0 PL=0
MOVL C01212 V=800.0 PL=0
MOVL C01213 V=800.0 PL=0
MOVL C01214 V=800.0 PL=0
MOVL C01215 V=800.0 PL=0
MOVL C01216 V=800.0 PL=0
MOVL C01217 V=800.0 PL=0
MOVL C01218 V=800.0 PL=0
MOVL C01219 V=800.0 PL=0
MOVL C01220 V=800.0 PL=0
MOVL C01221 V=800.0 PL=0
MOVL C01222 V=800.0 PL=0
MOVL C01223 V=800.0 PL=0
MOVL C01224 V=800.0 PL=0
MOVL C01225 V=800.0 PL=0
MOVL C01226 V=800.0 PL=0
MOVL C01227 V=800.0 PL=0
MOVL C01228 V=800.0 PL=0
MOVL C01229 V=800.0 PL=0
MOVL C01230 V=800.0 PL=0
MOVL C01231 V=800.0 PL=0
MOVL C01232 V=800.0 PL=0
MOVL C01233 V=800.0 PL=0
MOVL C01234 V=800.0 PL=0
MOVL C01235 V=800.0 PL=0
MOVL C01236 V=800.0 PL=0
MOVL C01237 V=800.0 PL=0
MOVL C01238 V=800.0 PL=0
MOVL C01239 V=800.0 PL=0
MOVL C01240 V=800.0 PL=0
MOVL C01241 V=800.0 PL=0
MOVL C01242 V=800.0 PL=0
MOVL C01243 V=800.0 PL=0
MOVL C01244 V=800.0 PL=0
MOVL C01245 V=800.0 PL=0
MOVL C01246 V=800.0 PL=0
MOVL C01247 V=800.0 PL=0
MOVL C01248 V=800.0 PL=0
MOVL C01249 V=800.0 PL=0
MOVL C01250 V=800.0 PL=0
MOVL C01251 V=800.0 PL=0
MOVL C01252 V=800.0 PL=0
MOVL C01253 V=800.0 PL=0
MOVL C01254 V=800.0 PL=0
MOVL C01255 V=800.0 PL=0
MOVL C01256 V=800.0 PL=0
MOVL C01257 V=800.0 PL=0
MOVL C01258 V=800.0 PL=0
MOVL C01259 V=800.0 PL=0
MOVL C01260 V=800.0 PL=0
MOVL C01261 V=800.0 PL=0
MOVL C01262 V=800.0 PL=0
MOVL C01263 V=800.0 PL=0
MOVL C01264 V=800.0 PL=0
MOVL C01265 V=800.0 PL=0
MOVL C01266 V=800.0 PL=0
MOVL C01267 V=800.0 PL=0
MOVL C01268 V=800.0 PL=0
MOVL C01269 V=800.0 PL=0
MOVL C01270 V=800.0 PL=0
MOVL C01271 V=800.0 PL=0
MOVL C01272 V=800.0 PL=0
MOVL C01273 V=800.0 PL=0
MOVL C01274 V=800.0 PL=0
MOVL C01275 V=800.0 PL=0
MOVL C01276 V=800.0 PL=0
MOVL C01277 V=800.0 PL=0
MOVL C01278 V=800.0 PL=0
MOVL C01279 V=800.0 PL=0
MOVL C01280 V=800.0 PL=0
MOVL C01281 V=800.0 PL=0
MOVL C01282 V=800.0 PL=0
MOVL C01283 V=800.0 PL=0
MOVL C01284 V=800.0 PL=0
MOVL C01285 V=800.0 PL=0
MOVL C01286 V=800.0 PL=0
MOVL C01287 V=800.0 PL=0
MOVL C01288 V=800.0 PL=0
MOVL C01289 V=800.0 PL=0
MOVL C01290 V=800.0 PL=0
MOVL C01291 V=800.0 PL=0
MOVL C01292 V=800.0 PL=0
MOVL C01293 V=800.0 PL=0
MOVL C01294 V=800.0 PL=0
MOVL C01295 V=800.0 PL=0
MOVL C01296 V=800.0 PL=0
MOVL C01297 V=800.0 PL=0
MOVL C01298 V=800.0 PL=0
MOVL C01299 V=800.0 PL=0
MOVL C01300 V=800.0 PL=0
MOVL C01301 V=800.0 PL=0
MOVL C01302 V=800.0 PL=0
MOVL C01303 V=800.0 PL=0
MOVL C01304 V=800.0 PL=0
MOVL C01305 V=800.0 PL=0
MOVL C01306 V=800.0 PL=0
MOVL C01307 V=800.0 PL=0
MOVL C01308 V=800.0 PL=0
MOVL C01309 V=800.0 PL=0
MOVL C01310 V=800.0 PL=0
MOVL C01311 V=800.0 PL=0
MOVL C01312 V=800.0 PL=0
MOVL C01313 V=800.0 PL=0
MOVL C01314 V=800.0 PL=0
MOVL C01315 V=800.0 PL=0
MOVL C01316 V=800.0 PL=0
MOVL C01317 V=800.0 PL=0
MOVL C01318 V=800.0 PL=0
MOVL C01319 V=800.0 PL=0
MOVL C01320 V=800.0 PL=0
MOVL C01321 V=800.0 PL=0
MOVL C01322 V=800.0 PL=0
MOVL C01323 V=800.0 PL=0
MOVL C01324 V=800.0 PL=0
MOVL C01325 V=800.0 PL=0
MOVL C01326 V=800.0 PL=0
MOVL C01327 V=800.0 PL=0
MOVL C01328 V=800.0 PL=0
MOVL C01329 V=800.0 PL=0
MOVL C01330 V=800.0 PL=0
MOVL C01331 V=800.0 PL=0
MOVL C01332 V=800.0 PL=0
MOVL C01333 V=800.0 PL=0
MOVL C01334 V=800.0 PL=0
MOVL C01335 V=800.0 PL=0
MOVL C01336 V=800.0 PL=0
MOVL C01337 V=800.0 PL=0
MOVL C01338 V=800.0 PL=0
MOVL C01339 V=800.0 PL=0
MOVL C01340 V=800.0 PL=0
MOVL C01341 V=800.0 PL=0
MOVL C01342 V=800.0 PL=0
MOVL C01343 V=800.0 PL=0
MOVL C01344 V=800.0 PL=0
MOVL C01345 V=800.0 PL=0
MOVL C01346 V=800.0 PL=0
MOVL C01347 V=800.0 PL=0
MOVL C01348 V=800.0 PL=0
MOVL C01349 V=800.0 PL=0
MOVL C01350 V=800.0 PL=0
MOVL C01351 V=800.0 PL=0
MOVL C01352 V=800.0 PL=0
MOVL C01353 V=800.0 PL=0
MOVL C01354 V=800.0 PL=0
MOVL C01355 V=800.0 PL=0
MOVL C01356 V=800.0 PL=0
MOVL C01357 V=800.0 PL=0
MOVL C01358 V=800.0 PL=0
MOVL C01359 V=800.0 PL=0
MOVL C01360 V=800.0 PL=0
MOVL C01361 V=800.0 PL=0
MOVL C01362 V=800.0 PL=0
MOVL C01363 V=800.0 PL=0
MOVL C01364 V=800.0 PL=0
MOVL C01365 V=800.0 PL=0
MOVL C01366 V=800.0 PL=0
MOVL C01367 V=800.0 PL=0
MOVL C01368 V=800.0 PL=0
MOVL C01369 V=800.0 PL=0
MOVL C01370 V=800.0 PL=0
MOVL C01371 V=800.0 PL=0
MOVL C01372 V=800.0 PL=0
MOVL C01373 V=800.0 PL=0
MOVL C01374 V=800.0 PL=0
MOVL C01375 V=800.0 PL=0
MOVL C01376 V=800.0 PL=0
MOVL C01377 V=800.0 PL=0
MOVL C01378 V=800.0 PL=0
MOVL C01379 V=800.0 PL=0
MOVL C01380 V=800.0 PL=0
MOVL C01381 V=800.0 PL=0
MOVL C01382 V=800.0 PL=0
MOVL C01383 V=800.0 PL=0
MOVL C01384 V=800.0 PL=0
MOVL C01385 V=800.0 PL=0
MOVL C01386 V=800.0 PL=0
MOVL C01387 V=800.0 PL=0
MOVL C01388 V=800.0 PL=0
MOVL C01389 V=800.0 PL=0
MOVL C01390 V=800.0 PL=0
MOVL C01391 V=800.0 PL=0
MOVL C01392 V=800.0 PL=0
MOVL C01393 V=800.0 PL=0
MOVL C01394 V=800.0 PL=0
MOVL C01395 V=800.0 PL=0
MOVL C01396 V=800.0 PL=0
MOVL C01397 V=800.0 PL=0
MOVL C01398 V=800.0 PL=0
MOVL C01399 V=800.0 PL=0
MOVL C01400 V=800.0 PL=0
MOVL C01401 V=800.0 PL=0
MOVL C01402 V=800.0 PL=0
MOVL C01403 V=800.0 PL=0
MOVL C01404 V=800.0 PL=0
MOVL C01405 V=800.0 PL=0
MOVL C01406 V=800.0 PL=0
MOVL C01407 V=800.0 PL=0
MOVL C01408 V=800.0 PL=0
MOVL C01409 V=800.0 PL=0
MOVL C01410 V=800.0 PL=0
MOVL C01411 V=800.0 PL=0
MOVL C01412 V=800.0 PL=0
MOVL C01413 V=800.0 PL=0
MOVL C01414 V=800.0 PL=0
MOVL C01415 V=800.0 PL=0
MOVL C01416 V=800.0 PL=0
MOVL C01417 V=800.0 PL=0
MOVL C01418 V=800.0 PL=0
MOVL C01419 V=800.0 PL=0
MOVL C01420 V=800.0 PL=0
MOVL C01421 V=800.0 PL=0
MOVL C01422 V=800.0 PL=0
MOVL C01423 V=800.0 PL=0
MOVL C01424 V=800.0 PL=0
MOVL C01425 V=800.0 PL=0
MOVL C01426 V=800.0 PL=0
MOVL C01427 V=800.0 PL=0
MOVL C01428 V=800.0 PL=0
MOVL C01429 V=800.0 PL=0
MOVL C01430 V=800.0 PL=0
MOVL C01431 V=800.0 PL=0
MOVL C01432 V=800.0 PL=0
MOVL C01433 V=800.0 PL=0
MOVL C01434 V=800.0 PL=0
MOVL C01435 V=800.0 PL=0
MOVL C01436 V=800.0 PL=0
MOVL C01437 V=800.0 PL=0
MOVL C01438 V=800.0 PL=0
MOVL C01439 V=800.0 PL=0
MOVL C01440 V=800.0 PL=0
MOVL C01441 V=800.0 PL=0
MOVL C01442 V=800.0 PL=0
MOVL C01443 V=800.0 PL=0
MOVL C01444 V=800.0 PL=0
MOVL C01445 V=800.0 PL=0
MOVL C01446 V=800.0 PL=0
MOVL C01447 V=800.0 PL=0
MOVL C01448 V=800.0 PL=0
MOVL C01449 V=800.0 PL=0
MOVL C01450 V=800.0 PL=0
MOVL C01451 V=800.0 PL=0
MOVL C01452 V=800.0 PL=0
MOVL C01453 V=800.0 PL=0
MOVL C01454 V=800.0 PL=0
MOVL C01455 V=800.0 PL=0
MOVL C01456 V=800.0 PL=0
MOVL C01457 V=800.0 PL=0
MOVL C01458 V=800.0 PL=0
MOVL C01459 V=800.0 PL=0
MOVL C01460 V=800.0 PL=0
MOVL C01461 V=800.0 PL=0
MOVL C01462 V=800.0 PL=0
MOVL C01463 V=800.0 PL=0
MOVL C01464 V=800.0 PL=0
MOVL C01465 V=800.0 PL=0
MOVL C01466 V=800.0 PL=0
MOVL C01467 V=800.0 PL=0
MOVL C01468 V=800.0 PL=0
MOVL C01469 V=800.0 PL=0
MOVL C01470 V=800.0 PL=0
MOVL C01471 V=800.0 PL=0
MOVL C01472 V=800.0 PL=0
MOVL C01473 V=800.0 PL=0
MOVL C01474 V=800.0 PL=0
MOVL C01475 V=800.0 PL=0
MOVL C01476 V=800.0 PL=0
MOVL C01477 V=800.0 PL=0
MOVL C01478 V=800.0 PL=0
MOVL C01479 V=800.0 PL=0
MOVL C01480 V=800.0 PL=0
MOVL C01481 V=800.0 PL=0
MOVL C01482 V=800.0 PL=0
MOVL C01483 V=800.0 PL=0
MOVL C01484 V=800.0 PL=0
MOVL C01485 V=800.0 PL=0
MOVL C01486 V=800.0 PL=0
MOVL C01487 V=800.0 PL=0
MOVL C01488 V=800.0 PL=0
MOVL C01489 V=800.0 PL=0
MOVL C01490 V=800.0 PL=0
MOVL C01491 V=800.0 PL=0
MOVL C01492 V=800.0 PL=0
MOVL C01493 V=800.0 PL=0
MOVL C01494 V=800.0 PL=0
MOVL C01495 V=800.0 PL=0
MOVL C01496 V=800.0 PL=0
MOVL C01497 V=800.0 PL=0
MOVL C01498 V=800.0 PL=0
MOVL C01499 V=800.0 PL=0
MOVL C01500 V=800.0 PL=0
MOVL C01501 V=800.0 PL=0
MOVL C01502 V=800.0 PL=0
MOVL C01503 V=800.0 PL=0
MOVL C01504 V=800.0 PL=0
MOVL C01505 V=800.0 PL=0
MOVL C01506 V=800.0 PL=0
MOVL C01507 V=800.0 PL=0
MOVL C01508 V=800.0 PL=0
MOVL C01509 V=800.0 PL=0
MOVL C01510 V=800.0 PL=0
MOVL C01511 V=800.0 PL=0
MOVL C01512 V=800.0 PL=0
MOVL C01513 V=800.0 PL=0
MOVL C01514 V=800.0 PL=0
MOVL C01515 V=800.0 PL=0
MOVL C01516 V=800.0 PL=0
MOVL C01517 V=800.0 PL=0
MOVL C01518 V=800.0 PL=0
MOVL C01519 V=800.0 PL=0
MOVL C01520 V=800.0 PL=0
MOVL C01521 V=800.0 PL=0
MOVL C01522 V=800.0 PL=0
MOVL C01523 V=800.0 PL=0
MOVL C01524 V=800.0 PL=0
MOVL C01525 V=800.0 PL=0
MOVL C01526 V=800.0 PL=0
MOVL C01527 V=800.0 PL=0
MOVL C01528 V=800.0 PL=0
MOVL C01529 V=800.0 PL=0
MOVL C01530 V=800.0 PL=0
MOVL C01531 V=800.0 PL=0
MOVL C01532 V=800.0 PL=0
MOVL C01533 V=800.0 PL=0
MOVL C01534 V=800.0 PL=0
MOVL C01535 V=800.0 PL=0
MOVL C01536 V=800.0 PL=0
MOVL C01537 V=800.0 PL=0
MOVL C01538 V=800.0 PL=0
MOVL C01539 V=800.0 PL=0
MOVL C01540 V=800.0 PL=0
MOVL C01541 V=800.0 PL=0
MOVL C01542 V=800.0 PL=0
MOVL C01543 V=800.0 PL=0
MOVL C01544 V=800.0 PL=0
MOVL C01545 V=800.0 PL=0
MOVL C01546 V=800.0 PL=0
MOVL C01547 V=800.0 PL=0
MOVL C01548 V=800.0 PL=0
MOVL C01549 V=800.0 PL=0
MOVL C01550 V=800.0 PL=0
MOVL C01551 V=800.0 PL=0
MOVL C01552 V=800.0 PL=0
MOVL C01553 V=800.0 PL=0
MOVL C01554 V=800.0 PL=0
MOVL C01555 V=800.0 PL=0
MOVL C01556 V=800.0 PL=0
MOVL C01557 V=800.0 PL=0
MOVL C01558 V=800.0 PL=0
MOVL C01559 V=800.0 PL=0
MOVL C01560 V=800.0 PL=0
MOVL C01561 V=800.0 PL=0
MOVL C01562 V=800.0 PL=0
MOVL C01563 V=800.0 PL=0
MOVL C01564 V=800.0 PL=0
MOVL C01565 V=800.0 PL=0
MOVL C01566 V=800.0 PL=0
MOVL C01567 V=800.0 PL=0
MOVL C01568 V=800.0 PL=0
MOVL C01569 V=800.0 PL=0
MOVL C01570 V=800.0 PL=0
MOVL C01571 V=800.0 PL=0
MOVL C01572 V=800.0 PL=0
MOVL C01573 V=800.0 PL=0
MOVL C01574 V=800.0 PL=0
MOVL C01575 V=800.0 PL=0
MOVL C01576 V=800.0 PL=0
MOVL C01577 V=800.0 PL=0
MOVL C01578 V=800.0 PL=0
MOVL C01579 V=800.0 PL=0
MOVL C01580 V=800.0 PL=0
MOVL C01581 V=800.0 PL=0
MOVL C01582 V=800.0 PL=0
MOVL C01583 V=800.0 PL=0
MOVL C01584 V=800.0 PL=0
MOVL C01585 V=800.0 PL=0
MOVL C01586 V=800.0 PL=0
MOVL C01587 V=800.0 PL=0
MOVL C01588 V=800.0 PL=0
MOVL C01589 V=800.0 PL=0
MOVL C01590 V=800.0 PL=0
MOVL C01591 V=800.0 PL=0
MOVL C01592 V=800.0 PL=0
MOVL C01593 V=800.0 PL=0
MOVL C01594 V=800.0 PL=0
MOVL C01595 V=800.0 PL=0
MOVL C01596 V=800.0 PL=0
MOVL C01597 V=800.0 PL=0
MOVL C01598 V=800.0 PL=0
MOVL C01599 V=800.0 PL=0
MOVL C01600 V=800.0 PL=0
MOVL C01601 V=800.0 PL=0
MOVL C01602 V=800.0 PL=0
MOVL C01603 V=800.0 PL=0
MOVL C01604 V=800.0 PL=0
MOVL C01605 V=800.0 PL=0
MOVL C01606 V=800.0 PL=0
MOVL C01607 V=800.0 PL=0
MOVL C01608 V=800.0 PL=0
MOVL C01609 V=800.0 PL=0
MOVL C01610 V=800.0 PL=0
MOVL C01611 V=800.0 PL=0
MOVL C01612 V=800.0 PL=0
MOVL C01613 V=800.0 PL=0
MOVL C01614 V=800.0 PL=0
MOVL C01615 V=800.0 PL=0
MOVL C01616 V=800.0 PL=0
MOVL C01617 V=800.0 PL=0
MOVL C01618 V=800.0 PL=0
MOVL C01619 V=800.0 PL=0
MOVL C01620 V=800.0 PL=0
MOVL C01621 V=800.0 PL=0
MOVL C01622 V=800.0 PL=0
MOVL C01623 V=800.0 PL=0
MOVL C01624 V=800.0 PL=0
MOVL C01625 V=800.0 PL=0
MOVL C01626 V=800.0 PL=0
MOVL C01627 V=800.0 PL=0
MOVL C01628 V=800.0 PL=0
MOVL C01629 V=800.0 PL=0
MOVL C01630 V=800.0 PL=0
MOVL C01631 V=800.0 PL=0
MOVL C01632 V=800.0 PL=0
MOVL C01633 V=800.0 PL=0
MOVL C01634 V=800.0 PL=0
MOVL C01635 V=800.0 PL=0
MOVL C01636 V=800.0 PL=0
MOVL C01637 V=800.0 PL=0
MOVL C01638 V=800.0 PL=0
MOVL C01639 V=800.0 PL=0
MOVL C01640 V=800.0 PL=0
MOVL C01641 V=800.0 PL=0
MOVL C01642 V=800.0 PL=0
MOVL C01643 V=800.0 PL=0
MOVL C01644 V=800.0 PL=0
MOVL C01645 V=800.0 PL=0
MOVL C01646 V=800.0 PL=0
MOVL C01647 V=800.0 PL=0
MOVL C01648 V=800.0 PL=0
MOVL C01649 V=800.0 PL=0
MOVL C01650 V=800.0 PL=0
MOVL C01651 V=800.0 PL=0
MOVL C01652 V=800.0 PL=0
MOVL C01653 V=800.0 PL=0
MOVL C01654 V=800.0 PL=0
MOVL C01655 V=800.0 PL=0
MOVL C01656 V=800.0 PL=0
MOVL C01657 V=800.0 PL=0
MOVL C01658 V=800.0 PL=0
MOVL C01659 V=800.0 PL=0
MOVL C01660 V=800.0 PL=0
MOVL C01661 V=800.0 PL=0
MOVL C01662 V=800.0 PL=0
MOVL C01663 V=800.0 PL=0
MOVL C01664 V=800.0 PL=0
MOVL C01665 V=800.0 PL=0
MOVL C01666 V=800.0 PL=0
MOVL C01667 V=800.0 PL=0
MOVL C01668 V=800.0 PL=0
MOVL C01669 V=800.0 PL=0
MOVL C01670 V=800.0 PL=0
MOVL C01671 V=800.0 PL=0
MOVL C01672 V=800.0 PL=0
MOVL C01673 V=800.0 PL=0
MOVL C01674 V=800.0 PL=0
MOVL C01675 V=800.0 PL=0
MOVL C01676 V=800.0 PL=0
MOVL C01677 V=800.0 PL=0
MOVL C01678 V=800.0 PL=0
MOVL C01679 V=800.0 PL=0
MOVL C01680 V=800.0 PL=0
MOVL C01681 V=800.0 PL=0
MOVL C01682 V=800.0 PL=0
MOVL C01683 V=800.0 PL=0
MOVL C01684 V=800.0 PL=0
MOVL C01685 V=800.0 PL=0
MOVL C01686 V=800.0 PL=0
MOVL C01687 V=800.0 PL=0
MOVL C01688 V=800.0 PL=0
MOVL C01689 V=800.0 PL=0
MOVL C01690 V=800.0 PL=0
MOVL C01691 V=800.0 PL=0
MOVL C01692 V=800.0 PL=0
MOVL C01693 V=800.0 PL=0
MOVL C01694 V=800.0 PL=0
MOVL C01695 V=800.0 PL=0
MOVL C01696 V=800.0 PL=0
MOVL C01697 V=800.0 PL=0
MOVL C01698 V=800.0 PL=0
MOVL C01699 V=800.0 PL=0
MOVL C01700 V=800.0 PL=0
MOVL C01701 V=800.0 PL=0
MOVL C01702 V=800.0 PL=0
MOVL C01703 V=800.0 PL=0
MOVL C01704 V=800.0 PL=0
MOVL C01705 V=800.0 PL=0
MOVL C01706 V=800.0 PL=0
MOVL C01707 V=800.0 PL=0
MOVL C01708 V=800.0 PL=0
MOVL C01709 V=800.0 PL=0
MOVL C01710 V=800.0 PL=0
MOVL C01711 V=800.0 PL=0
MOVL C01712 V=800.0 PL=0
MOVL C01713 V=800.0 PL=0
MOVL C01714 V=800.0 PL=0
MOVL C01715 V=800.0 PL=0
MOVL C01716 V=800.0 PL=0
MOVL C01717 V=800.0 PL=0
MOVL C01718 V=800.0 PL=0
MOVL C01719 V=800.0 PL=0
MOVL C01720 V=800.0 PL=0
MOVL C01721 V=800.0 PL=0
MOVL C01722 V=800.0 PL=0
MOVL C01723 V=800.0 PL=0
MOVL C01724 V=800.0 PL=0
MOVL C01725 V=800.0 PL=0
MOVL C01726 V=800.0 PL=0
MOVL C01727 V=800.0 PL=0
MOVL C01728 V=800.0 PL=0
MOVL C01729 V=800.0 PL=0
MOVL C01730 V=800.0 PL=0
MOVL C01731 V=800.0 PL=0
MOVL C01732 V=800.0 PL=0
MOVL C01733 V=800.0 PL=0
MOVL C01734 V=800.0 PL=0
MOVL C01735 V=800.0 PL=0
MOVL C01736 V=800.0 PL=0
MOVL C01737 V=800.0 PL=0
MOVL C01738 V=800.0 PL=0
MOVL C01739 V=800.0 PL=0
MOVL C01740 V=800.0 PL=0
MOVL C01741 V=800.0 PL=0
MOVL C01742 V=800.0 PL=0
MOVL C01743 V=800.0 PL=0
MOVL C01744 V=800.0 PL=0
MOVL C01745 V=800.0 PL=0
MOVL C01746 V=800.0 PL=0
MOVL C01747 V=800.0 PL=0
MOVL C01748 V=800.0 PL=0
MOVL C01749 V=800.0 PL=0
MOVL C01750 V=800.0 PL=0
MOVL C01751 V=800.0 PL=0
MOVL C01752 V=800.0 PL=0
MOVL C01753 V=800.0 PL=0
MOVL C01754 V=800.0 PL=0
MOVL C01755 V=800.0 PL=0
MOVL C01756 V=800.0 PL=0
MOVL C01757 V=800.0 PL=0
MOVL C01758 V=800.0 PL=0
MOVL C01759 V=800.0 PL=0
MOVL C01760 V=800.0 PL=0
MOVL C01761 V=800.0 PL=0
MOVL C01762 V=800.0 PL=0
MOVL C01763 V=800.0 PL=0
MOVL C01764 V=800.0 PL=0
MOVL C01765 V=800.0 PL=0
MOVL C01766 V=800.0 PL=0
MOVL C01767 V=800.0 PL=0
MOVL C01768 V=800.0 PL=0
MOVL C01769 V=800.0 PL=0
MOVL C01770 V=800.0 PL=0
MOVL C01771 V=800.0 PL=0
MOVL C01772 V=800.0 PL=0
MOVL C01773 V=800.0 PL=0
MOVL C01774 V=800.0 PL=0
MOVL C01775 V=800.0 PL=0
MOVL C01776 V=800.0 PL=0
MOVL C01777 V=800.0 PL=0
MOVL C01778 V=800.0 PL=0
MOVL C01779 V=800.0 PL=0
MOVL C01780 V=800.0 PL=0
MOVL C01781 V=800.0 PL=0
MOVL C01782 V=800.0 PL=0
MOVL C01783 V=800.0 PL=0
MOVL C01784 V=800.0 PL=0
MOVL C01785 V=800.0 PL=0
MOVL C01786 V=800.0 PL=0
MOVL C01787 V=800.0 PL=0
MOVL C01788 V=800.0 PL=0
MOVL C01789 V=800.0 PL=0
MOVL C01790 V=800.0 PL=0
MOVL C01791 V=800.0 PL=0
MOVL C01792 V=800.0 PL=0
MOVL C01793 V=800.0 PL=0
MOVL C01794 V=800.0 PL=0
MOVL C01795 V=800.0 PL=0
MOVL C01796 V=800.0 PL=0
MOVL C01797 V=800.0 PL=0
MOVL C01798 V=800.0 PL=0
MOVL C01799 V=800.0 PL=0
MOVL C01800 V=800.0 PL=0
MOVL C01801 V=800.0 PL=0
MOVL C01802 V=800.0 PL=0
MOVL C01803 V=800.0 PL=0
MOVL C01804 V=800.0 PL=0
MOVL C01805 V=800.0 PL=0
MOVL C01806 V=800.0 PL=0
MOVL C01807 V=800.0 PL=0
MOVL C01808 V=800.0 PL=0
MOVL C01809 V=800.0 PL=0
MOVL C01810 V=800.0 PL=0
MOVL C01811 V=800.0 PL=0
MOVL C01812 V=800.0 PL=0
MOVL C01813 V=800.0 PL=0
MOVL C01814 V=800.0 PL=0
MOVL C01815 V=800.0 PL=0
MOVL C01816 V=800.0 PL=0
MOVL C01817 V=800.0 PL=0
MOVL C01818 V=800.0 PL=0
MOVL C01819 V=800.0 PL=0
MOVL C01820 V=800.0 PL=0
MOVL C01821 V=800.0 PL=0
MOVL C01822 V=800.0 PL=0
MOVL C01823 V=800.0 PL=0
MOVL C01824 V=800.0 PL=0
MOVL C01825 V=800.0 PL=0
MOVL C01826 V=800.0 PL=0
MOVL C01827 V=800.0 PL=0
MOVL C01828 V=800.0 PL=0
MOVL C01829 V=800.0 PL=0
MOVL C01830 V=800.0 PL=0
MOVL C01831 V=800.0 PL=0
MOVL C01832 V=800.0 PL=0
MOVL C01833 V=800.0 PL=0
MOVL C01834 V=800.0 PL=0
MOVL C01835 V=800.0 PL=0
MOVL C01836 V=800.0 PL=0
MOVL C01837 V=800.0 PL=0
MOVL C01838 V=800.0 PL=0
MOVL C01839 V=800.0 PL=0
MOVL C01840 V=800.0 PL=0
MOVL C01841 V=800.0 PL=0
MOVL C01842 V=800.0 PL=0
MOVL C01843 V=800.0 PL=0
MOVL C01844 V=800.0 PL=0
MOVL C01845 V=800.0 PL=0
MOVL C01846 V=800.0 PL=0
MOVL C01847 V=800.0 PL=0
MOVL C01848 V=800.0 PL=0
MOVL C01849 V=800.0 PL=0
MOVL C01850 V=800.0 PL=0
MOVL C01851 V=800.0 PL=0
MOVL C01852 V=800.0 PL=0
MOVL C01853 V=800.0 PL=0
MOVL C01854 V=800.0 PL=0
MOVL C01855 V=800.0 PL=0
MOVL C01856 V=800.0 PL=0
MOVL C01857 V=800.0 PL=0
MOVL C01858 V=800.0 PL=0
MOVL C01859 V=800.0 PL=0
MOVL C01860 V=800.0 PL=0
MOVL C01861 V=800.0 PL=0
MOVL C01862 V=800.0 PL=0
MOVL C01863 V=800.0 PL=0
MOVL C01864 V=800.0 PL=0
MOVL C01865 V=800.0 PL=0
MOVL C01866 V=800.0 PL=0
MOVL C01867 V=800.0 PL=0
MOVL C01868 V=800.0 PL=0
MOVL C01869 V=800.0 PL=0
MOVL C01870 V=800.0 PL=0
MOVL C01871 V=800.0 PL=0
MOVL C01872 V=800.0 PL=0
MOVL C01873 V=800.0 PL=0
MOVL C01874 V=800.0 PL=0
MOVL C01875 V=800.0 PL=0
MOVL C01876 V=800.0 PL=0
MOVL C01877 V=800.0 PL=0
MOVL C01878 V=800.0 PL=0
MOVL C01879 V=800.0 PL=0
MOVL C01880 V=800.0 PL=0
MOVL C01881 V=800.0 PL=0
MOVL C01882 V=800.0 PL=0
MOVL C01883 V=800.0 PL=0
MOVL C01884 V=800.0 PL=0
MOVL C01885 V=800.0 PL=0
MOVL C01886 V=800.0 PL=0
MOVL C01887 V=800.0 PL=0
MOVL C01888 V=800.0 PL=0
MOVL C01889 V=800.0 PL=0
MOVL C01890 V=800.0 PL=0
MOVL C01891 V=800.0 PL=0
MOVL C01892 V=800.0 PL=0
MOVL C01893 V=800.0 PL=0
MOVL C01894 V=800.0 PL=0
MOVL C01895 V=800.0 PL=0
MOVL C01896 V=800.0 PL=0
MOVL C01897 V=800.0 PL=0
MOVL C01898 V=800.0 PL=0
MOVL C01899 V=800.0 PL=0
MOVL C01900 V=800.0 PL=0
MOVL C01901 V=800.0 PL=0
MOVL C01902 V=800.0 PL=0
MOVL C01903 V=800.0 PL=0
MOVL C01904 V=800.0 PL=0
MOVL C01905 V=800.0 PL=0
MOVL C01906 V=800.0 PL=0
MOVL C01907 V=800.0 PL=0
MOVL C01908 V=800.0 PL=0
MOVL C01909 V=800.0 PL=0
MOVL C01910 V=800.0 PL=0
MOVL C01911 V=800.0 PL=0
MOVL C01912 V=800.0 PL=0
MOVL C01913 V=800.0 PL=0
MOVL C01914 V=800.0 PL=0
MOVL C01915 V=800.0 PL=0
MOVL C01916 V=800.0 PL=0
MOVL C01917 V=800.0 PL=0
MOVL C01918 V=800.0 PL=0
MOVL C01919 V=800.0 PL=0
MOVL C01920 V=800.0 PL=0
MOVL C01921 V=800.0 PL=0
MOVL C01922 V=800.0 PL=0
MOVL C01923 V=800.0 PL=0
MOVL C01924 V=800.0 PL=0
MOVL C01925 V=800.0 PL=0
MOVL C01926 V=800.0 PL=0
MOVL C01927 V=800.0 PL=0
MOVL C01928 V=800.0 PL=0
MOVL C01929 V=800.0 PL=0
MOVL C01930 V=800.0 PL=0
MOVL C01931 V=800.0 PL=0
MOVL C01932 V=800.0 PL=0
MOVL C01933 V=800.0 PL=0
MOVL C01934 V=800.0 PL=0
MOVL C01935 V=800.0 PL=0
MOVL C01936 V=800.0 PL=0
MOVL C01937 V=800.0 PL=0
MOVL C01938 V=800.0 PL=0
MOVL C01939 V=800.0 PL=0
MOVL C01940 V=800.0 PL=0
MOVL C01941 V=800.0 PL=0
MOVL C01942 V=800.0 PL=0
MOVL C01943 V=800.0 PL=0
MOVL C01944 V=800.0 PL=0
MOVL C01945 V=800.0 PL=0
MOVL C01946 V=800.0 PL=0
MOVL C01947 V=800.0 PL=0
MOVL C01948 V=800.0 PL=0
MOVL C01949 V=800.0 PL=0
MOVL C01950 V=800.0 PL=0
MOVL C01951 V=800.0 PL=0
MOVL C01952 V=800.0 PL=0
MOVL C01953 V=800.0 PL=0
MOVL C01954 V=800.0 PL=0
MOVL C01955 V=800.0 PL=0
MOVL C01956 V=800.0 PL=0
MOVL C01957 V=800.0 PL=0
MOVL C01958 V=800.0 PL=0
MOVL C01959 V=800.0 PL=0
MOVL C01960 V=800.0 PL=0
MOVL C01961 V=800.0 PL=0
MOVL C01962 V=800.0 PL=0
MOVL C01963 V=800.0 PL=0
MOVL C01964 V=800.0 PL=0
MOVL C01965 V=800.0 PL=0
MOVL C01966 V=800.0 PL=0
MOVL C01967 V=800.0 PL=0
MOVL C01968 V=800.0 PL=0
MOVL C01969 V=800.0 PL=0
MOVL C01970 V=800.0 PL=0
MOVL C01971 V=800.0 PL=0
MOVL C01972 V=800.0 PL=0
MOVL C01973 V=800.0 PL=0
MOVL C01974 V=800.0 PL=0
MOVL C01975 V=800.0 PL=0
MOVL C01976 V=800.0 PL=0
MOVL C01977 V=800.0 PL=0
MOVL C01978 V=800.0 PL=0
MOVL C01979 V=800.0 PL=0
MOVL C01980 V=800.0 PL=0
MOVL C01981 V=800.0 PL=0
MOVL C01982 V=800.0 PL=0
MOVL C01983 V=800.0 PL=0
MOVL C01984 V=800.0 PL=0
MOVL C01985 V=800.0 PL=0
MOVL C01986 V=800.0 PL=0
MOVL C01987 V=800.0 PL=0
MOVL C01988 V=800.0 PL=0
MOVL C01989 V=800.0 PL=0
MOVL C01990 V=800.0 PL=0
MOVL C01991 V=800.0 PL=0
MOVL C01992 V=800.0 PL=0
MOVL C01993 V=800.0 PL=0
MOVL C01994 V=800.0 PL=0
MOVL C01995 V=800.0 PL=0
MOVL C01996 V=800.0 PL=0
MOVL C01997 V=800.0 PL=0
MOVL C01998 V=800.0 PL=0
MOVL C01999 V=800.0 PL=0
MOVL C02000 V=800.0 PL=0
MOVL C02001 V=800.0 PL=0
MOVL C02002 V=800.0 PL=0
MOVL C02003 V=800.0 PL=0
MOVL C02004 V=800.0 PL=0
MOVL C02005 V=800.0 PL=0
MOVL C02006 V=800.0 PL=0
MOVL C02007 V=800.0 PL=0
MOVL C02008 V=800.0 PL=0
MOVL C02009 V=800.0 PL=0
MOVL C02010 V=800.0 PL=0
MOVL C02011 V=800.0 PL=0
MOVL C02012 V=800.0 PL=0
MOVL C02013 V=800.0 PL=0
MOVL C02014 V=800.0 PL=0
MOVL C02015 V=800.0 PL=0
MOVL C02016 V=800.0 PL=0
MOVL C02017 V=800.0 PL=0
MOVL C02018 V=800.0 PL=0
MOVL C02019 V=800.0 PL=0
MOVL C02020 V=800.0 PL=0
MOVL C02021 V=800.0 PL=0
MOVL C02022 V=800.0 PL=0
MOVL C02023 V=800.0 PL=0
MOVL C02024 V=800.0 PL=0
MOVL C02025 V=800.0 PL=0
MOVL C02026 V=800.0 PL=0
MOVL C02027 V=800.0 PL=0
MOVL C02028 V=800.0 PL=0
MOVL C02029 V=800.0 PL=0
MOVL C02030 V=800.0 PL=0
MOVL C02031 V=800.0 PL=0
MOVL C02032 V=800.0 PL=0
MOVL C02033 V=800.0 PL=0
MOVL C02034 V=800.0 PL=0
MOVL C02035 V=800.0 PL=0
MOVL C02036 V=800.0 PL=0
MOVL C02037 V=800.0 PL=0
MOVL C02038 V=800.0 PL=0
MOVL C02039 V=800.0 PL=0
MOVL C02040 V=800.0 PL=0
MOVL C02041 V=800.0 PL=0
MOVL C02042 V=800.0 PL=0
MOVL C02043 V=800.0 PL=0
MOVL C02044 V=800.0 PL=0
MOVL C02045 V=800.0 PL=0
MOVL C02046 V=800.0 PL=0
